LIN {X 0,Y 248.769,Z 1005.47,A -85,B 0,C 180,E1 11445.151,E2 11445.151} C_VEL
LIN {X 0,Y 248.089,Z 1009.313,A -85,B 0,C 180,E1 11439.986,E2 11439.986} C_VEL
LIN {X 0,Y 247.98,Z 1011.318,A -85,B 0,C 180,E1 11435.56,E2 11435.56} C_VEL
LIN {X 0,Y 248.003,Z 1012.187,A -85,B 0,C 180,E1 11431.393,E2 11431.393} C_VEL
LIN {X 0,Y 247.976,Z 1011.971,A -85,B 0,C 180,E1 11426.771,E2 11426.771} C_VEL
LIN {X 0,Y 247.994,Z 1010.436,A -85,B 0,C 180,E1 11422.362,E2 11422.362} C_VEL
LIN {X 0,Y 248.248,Z 1007.938,A -85,B 0,C 180,E1 11418.154,E2 11418.154} C_VEL
LIN {X 0,Y 249.171,Z 1003.742,A -85,B 0,C 180,E1 11413.215,E2 11413.215} C_VEL
LIN {X 0,Y 251.144,Z 997.579,A -85,B 0,C 180,E1 11408.065,E2 11408.065} C_VEL
LIN {X 0,Y 254.45,Z 989.685,A -85,B 0,C 180,E1 11402.891,E2 11402.891} C_VEL
LIN {X 0,Y 258.825,Z 980.598,A -85,B 0,C 180,E1 11398.196,E2 11398.196} C_VEL
LIN {X 0,Y 264.874,Z 969.114,A -85,B 0,C 180,E1 11393.396,E2 11393.396} C_VEL
LIN {X 0,Y 271.46,Z 957.155,A -85,B 0,C 180,E1 11389.323,E2 11389.323} C_VEL
LIN {X 0,Y 279.185,Z 943.15,A -85,B 0,C 180,E1 11385.428,E2 11385.428} C_VEL
LIN {X 0,Y 287.538,Z 927.889,A -85,B 0,C 180,E1 11381.926,E2 11381.926} C_VEL
LIN {X 0,Y 296.257,Z 911.009,A -85,B 0,C 180,E1 11378.787,E2 11378.787} C_VEL
LIN {X 0,Y 305.508,Z 892.125,A -85,B 0,C 180,E1 11375.916,E2 11375.916} C_VEL
LIN {X 0,Y 313.91,Z 873.62,A -85,B 0,C 180,E1 11373.613,E2 11373.613} C_VEL
LIN {X 0,Y 321.806,Z 854.322,A -85,B 0,C 180,E1 11371.658,E2 11371.658} C_VEL
LIN {X 0,Y 329.269,Z 834.233,A -85,B 0,C 180,E1 11369.98,E2 11369.98} C_VEL
LIN {X 0,Y 335.891,Z 813.522,A -85,B 0,C 180,E1 11368.596,E2 11368.596} C_VEL
LIN {X 0,Y 341.852,Z 792.201,A -85,B 0,C 180,E1 11367.446,E2 11367.446} C_VEL
LIN {X 0,Y 346.788,Z 770.459,A -85,B 0,C 180,E1 11366.544,E2 11366.544} C_VEL
LIN {X 0,Y 351.119,Z 746.303,A -85,B 0,C 180,E1 11365.792,E2 11365.792} C_VEL
LIN {X 0,Y 353.796,Z 723.704,A -85,B 0,C 180,E1 11365.251,E2 11365.251} C_VEL
LIN {X 0,Y 369.048,Z 537.52,A -85,B 0,C 180,E1 11361.492,E2 11361.492} C_VEL
LIN {X 0,Y 363.248,Z 527.675,A -85,B 0,C 180,E1 11359.036,E2 11359.036} C_VEL
LIN {X 0,Y 357.672,Z 518.823,A -85,B 0,C 180,E1 11356.441,E2 11356.441} C_VEL
LIN {X 0,Y 350.936,Z 509.322,A -85,B 0,C 180,E1 11352.923,E2 11352.923} C_VEL
LIN {X 0,Y 346.797,Z 503.841,A -85,B 0,C 180,E1 11350.464,E2 11350.464} C_VEL
LIN {X 0,Y 343.075,Z 498.85,A -85,B 0,C 180,E1 11347.957,E2 11347.957} C_VEL
LIN {X 0,Y 339.371,Z 493.892,A -85,B 0,C 180,E1 11345.07,E2 11345.07} C_VEL
LIN {X 0,Y 336.137,Z 489.935,A -85,B 0,C 180,E1 11342.114,E2 11342.114} C_VEL
LIN {X 0,Y 335.121,Z 488.35,A -85,B 0,C 180,E1 11341.025,E2 11341.025} C_VEL
LIN {X 0,Y 331.973,Z 484.932,A -85,B 0,C 180,E1 11337.151,E2 11337.151} C_VEL
LIN {X 0,Y 330.953,Z 482.618,A -85,B 0,C 180,E1 11335.32,E2 11335.32} C_VEL
LIN {X 0,Y 328.272,Z 480.723,A -85,B 0,C 180,E1 11328.224,E2 11328.224} C_VEL
LIN {X 0,Y 328.227,Z 480.713,A -85,B 0,C 180,E1 11323.36,E2 11323.36} C_VEL
LIN {X 0,Y 330.956,Z 482.61,A -85,B 0,C 180,E1 11315.929,E2 11315.929} C_VEL
LIN {X 0,Y 333.571,Z 487.051,A -85,B 0,C 180,E1 11311.926,E2 11311.926} C_VEL
LIN {X 0,Y 335.647,Z 488.946,A -85,B 0,C 180,E1 11309.683,E2 11309.683} C_VEL
LIN {X 0,Y 338.748,Z 493.298,A -85,B 0,C 180,E1 11306.701,E2 11306.701} C_VEL
LIN {X 0,Y 340.159,Z 494.956,A -85,B 0,C 180,E1 11305.539,E2 11305.539} C_VEL
LIN {X 0,Y 344.371,Z 500.521,A -85,B 0,C 180,E1 11302.421,E2 11302.421} C_VEL
LIN {X 0,Y 348.619,Z 506.23,A -85,B 0,C 180,E1 11299.71,E2 11299.71} C_VEL
LIN {X 0,Y 352.841,Z 512.104,A -85,B 0,C 180,E1 11297.314,E2 11297.314} C_VEL
LIN {X 0,Y 358.459,Z 519.986,A -85,B 0,C 180,E1 11294.489,E2 11294.489} C_VEL
LIN {X 0,Y 365.158,Z 529.934,A -85,B 0,C 180,E1 11291.493,E2 11291.493} C_VEL
LIN {X 0,Y 368.682,Z 535.581,A -85,B 0,C 180,E1 11290.037,E2 11290.037} C_VEL
LIN {X 0,Y 353.501,Z 718.347,A -85,B 0,C 180,E1 11286.344,E2 11286.344} C_VEL
LIN {X 0,Y 350.103,Z 742.254,A -85,B 0,C 180,E1 11285.689,E2 11285.689} C_VEL
LIN {X 0,Y 345.867,Z 764.626,A -85,B 0,C 180,E1 11284.859,E2 11284.859} C_VEL
LIN {X 0,Y 340.555,Z 786.357,A -85,B 0,C 180,E1 11283.797,E2 11283.797} C_VEL
LIN {X 0,Y 334.282,Z 808.106,A -85,B 0,C 180,E1 11282.465,E2 11282.465} C_VEL
LIN {X 0,Y 327.833,Z 827.172,A -85,B 0,C 180,E1 11281.019,E2 11281.019} C_VEL
LIN {X 0,Y 319.891,Z 847.961,A -85,B 0,C 180,E1 11279.098,E2 11279.098} C_VEL
LIN {X 0,Y 312.126,Z 866.095,A -85,B 0,C 180,E1 11277.05,E2 11277.05} C_VEL
LIN {X 0,Y 303.456,Z 884.529,A -85,B 0,C 180,E1 11274.522,E2 11274.522} C_VEL
LIN {X 0,Y 295.342,Z 900.625,A -85,B 0,C 180,E1 11271.856,E2 11271.856} C_VEL
LIN {X 0,Y 286.891,Z 916.302,A -85,B 0,C 180,E1 11268.694,E2 11268.694} C_VEL
LIN {X 0,Y 278.817,Z 930.785,A -85,B 0,C 180,E1 11265.169,E2 11265.169} C_VEL
LIN {X 0,Y 271.276,Z 943.789,A -85,B 0,C 180,E1 11261.258,E2 11261.258} C_VEL
LIN {X 0,Y 264.24,Z 956.093,A -85,B 0,C 180,E1 11256.729,E2 11256.729} C_VEL
LIN {X 0,Y 259.012,Z 965.539,A -85,B 0,C 180,E1 11252.427,E2 11252.427} C_VEL
LIN {X 0,Y 254.363,Z 974.561,A -85,B 0,C 180,E1 11247.29,E2 11247.29} C_VEL
LIN {X 0,Y 251.266,Z 981.545,A -85,B 0,C 180,E1 11242.247,E2 11242.247} C_VEL
LIN {X 0,Y 249.362,Z 986.687,A -85,B 0,C 180,E1 11237.253,E2 11237.253} C_VEL
LIN {X 0,Y 248.437,Z 990.344,A -85,B 0,C 180,E1 11232.425,E2 11232.425} C_VEL
LIN {X 0,Y 248.066,Z 992.682,A -85,B 0,C 180,E1 11227.373,E2 11227.373} C_VEL
LIN {X 0,Y 247.999,Z 993.543,A -85,B 0,C 180,E1 11223.409,E2 11223.409} C_VEL
LIN {X 0,Y 248.016,Z 993.556,A -85,B 0,C 180,E1 11219.465,E2 11219.465} C_VEL
LIN {X 0,Y 248.186,Z 992.42,A -85,B 0,C 180,E1 11214.534,E2 11214.534} C_VEL
LIN {X 0,Y 248.752,Z 989.887,A -85,B 0,C 180,E1 11209.667,E2 11209.667} C_VEL
LIN {X 0,Y 250.122,Z 986.016,A -85,B 0,C 180,E1 11204.631,E2 11204.631} C_VEL
LIN {X 0,Y 252.616,Z 980.364,A -85,B 0,C 180,E1 11199.475,E2 11199.475} C_VEL
LIN {X 0,Y 256.451,Z 973.276,A -85,B 0,C 180,E1 11194.426,E2 11194.426} C_VEL
LIN {X 0,Y 259.234,Z 968.524,A -85,B 0,C 180,E1 11191.656,E2 11191.656} C_VEL
LIN {X 0,Y 260.09,Z 965.887,A -85,B 0,C 180,E1 11190.056,E2 11190.056} C_VEL
LIN {X 0,Y 259.629,Z 958.618,A -85,B 0,C 180,E1 11185.651,E2 11185.651} C_VEL
LIN {X 0,Y 260.902,Z 955.846,A -85,B 0,C 180,E1 11184.347,E2 11184.347} C_VEL
LIN {X 0,Y 268.781,Z 944.21,A -85,B 0,C 180,E1 11180.014,E2 11180.014} C_VEL
LIN {X 0,Y 278.131,Z 930.421,A -85,B 0,C 180,E1 11175.856,E2 11175.856} C_VEL
LIN {X 0,Y 286.879,Z 917.067,A -85,B 0,C 180,E1 11172.591,E2 11172.591} C_VEL
LIN {X 0,Y 297.228,Z 900.535,A -85,B 0,C 180,E1 11169.293,E2 11169.293} C_VEL
LIN {X 0,Y 307.195,Z 883.613,A -85,B 0,C 180,E1 11166.542,E2 11166.542} C_VEL
LIN {X 0,Y 316.877,Z 865.511,A -85,B 0,C 180,E1 11164.163,E2 11164.163} C_VEL
LIN {X 0,Y 326.234,Z 846.492,A -85,B 0,C 180,E1 11162.108,E2 11162.108} C_VEL
LIN {X 0,Y 334.593,Z 827.332,A -85,B 0,C 180,E1 11160.429,E2 11160.429} C_VEL
LIN {X 0,Y 342.772,Z 806.039,A -85,B 0,C 180,E1 11158.914,E2 11158.914} C_VEL
LIN {X 0,Y 349.225,Z 786.548,A -85,B 0,C 180,E1 11157.799,E2 11157.799} C_VEL
LIN {X 0,Y 355.509,Z 763.656,A -85,B 0,C 180,E1 11156.762,E2 11156.762} C_VEL
LIN {X 0,Y 359.938,Z 743.618,A -85,B 0,C 180,E1 11156.062,E2 11156.062} C_VEL
LIN {X 0,Y 363.887,Z 719.388,A -85,B 0,C 180,E1 11155.435,E2 11155.435} C_VEL
LIN {X 0,Y 383.022,Z 548.711,A -85,B 0,C 180,E1 11151.972,E2 11151.972} C_VEL
LIN {X 0,Y 381.952,Z 546.067,A -85,B 0,C 180,E1 11150.508,E2 11150.508} C_VEL
LIN {X 0,Y 381.336,Z 544.156,A -85,B 0,C 180,E1 11149.272,E2 11149.272} C_VEL
LIN {X 0,Y 380.669,Z 542.357,A -85,B 0,C 180,E1 11146.172,E2 11146.172} C_VEL
LIN {X 0,Y 381.477,Z 544.535,A -85,B 0,C 180,E1 11142.851,E2 11142.851} C_VEL
LIN {X 0,Y 382.931,Z 548.576,A -85,B 0,C 180,E1 11140.555,E2 11140.555} C_VEL
LIN {X 0,Y 383.035,Z 549.077,A -85,B 0,C 180,E1 11140.399,E2 11140.399} C_VEL
LIN {X 0,Y 362.692,Z 730.721,A -85,B 0,C 180,E1 11136.705,E2 11136.705} C_VEL
LIN {X 0,Y 358.409,Z 754.445,A -85,B 0,C 180,E1 11136.093,E2 11136.093} C_VEL
LIN {X 0,Y 352.927,Z 777.381,A -85,B 0,C 180,E1 11135.333,E2 11135.333} C_VEL
LIN {X 0,Y 346.699,Z 798.517,A -85,B 0,C 180,E1 11134.399,E2 11134.399} C_VEL
LIN {X 0,Y 339.018,Z 820.594,A -85,B 0,C 180,E1 11133.152,E2 11133.152} C_VEL
LIN {X 0,Y 331.343,Z 839.865,A -85,B 0,C 180,E1 11131.787,E2 11131.787} C_VEL
LIN {X 0,Y 321.816,Z 861.077,A -85,B 0,C 180,E1 11129.921,E2 11129.921} C_VEL
LIN {X 0,Y 312.718,Z 879.494,A -85,B 0,C 180,E1 11127.925,E2 11127.925} C_VEL
LIN {X 0,Y 302.497,Z 898.396,A -85,B 0,C 180,E1 11125.396,E2 11125.396} C_VEL
LIN {X 0,Y 292.361,Z 916.045,A -85,B 0,C 180,E1 11122.502,E2 11122.502} C_VEL
LIN {X 0,Y 282.55,Z 932.109,A -85,B 0,C 180,E1 11119.232,E2 11119.232} C_VEL
LIN {X 0,Y 272.441,Z 948.205,A -85,B 0,C 180,E1 11115.201,E2 11115.201} C_VEL
LIN {X 0,Y 263.857,Z 961.864,A -85,B 0,C 180,E1 11110.969,E2 11110.969} C_VEL
LIN {X 0,Y 256.394,Z 973.776,A -85,B 0,C 180,E1 11106.359,E2 11106.359} C_VEL
LIN {X 0,Y 250.204,Z 984.397,A -85,B 0,C 180,E1 11101.306,E2 11101.306} C_VEL
LIN {X 0,Y 245.794,Z 992.731,A -85,B 0,C 180,E1 11096.328,E2 11096.328} C_VEL
LIN {X 0,Y 242.454,Z 1000.349,A -85,B 0,C 180,E1 11090.527,E2 11090.527} C_VEL
LIN {X 0,Y 240.859,Z 1005.238,A -85,B 0,C 180,E1 11085.621,E2 11085.621} C_VEL
LIN {X 0,Y 240.107,Z 1009.027,A -85,B 0,C 180,E1 11080.322,E2 11080.322} C_VEL
LIN {X 0,Y 239.985,Z 1011.028,A -85,B 0,C 180,E1 11075.746,E2 11075.746} C_VEL
LIN {X 0,Y 240.011,Z 1011.863,A -85,B 0,C 180,E1 11071.678,E2 11071.678} C_VEL
LIN {X 0,Y 239.993,Z 1011.753,A -85,B 0,C 180,E1 11067.381,E2 11067.381} C_VEL
LIN {X 0,Y 239.989,Z 1010.321,A -85,B 0,C 180,E1 11062.548,E2 11062.548} C_VEL
LIN {X 0,Y 240.269,Z 1007.717,A -85,B 0,C 180,E1 11057.936,E2 11057.936} C_VEL
LIN {X 0,Y 241.247,Z 1003.603,A -85,B 0,C 180,E1 11052.895,E2 11052.895} C_VEL
LIN {X 0,Y 243.357,Z 997.456,A -85,B 0,C 180,E1 11047.545,E2 11047.545} C_VEL
LIN {X 0,Y 246.843,Z 989.668,A -85,B 0,C 180,E1 11042.246,E2 11042.246} C_VEL
LIN {X 0,Y 251.412,Z 980.698,A -85,B 0,C 180,E1 11037.469,E2 11037.469} C_VEL
LIN {X 0,Y 257.831,Z 969.179,A -85,B 0,C 180,E1 11032.505,E2 11032.505} C_VEL
LIN {X 0,Y 264.721,Z 957.254,A -85,B 0,C 180,E1 11028.347,E2 11028.347} C_VEL
LIN {X 0,Y 272.787,Z 943.296,A -85,B 0,C 180,E1 11024.389,E2 11024.389} C_VEL
LIN {X 0,Y 281.465,Z 928.077,A -85,B 0,C 180,E1 11020.843,E2 11020.843} C_VEL
LIN {X 0,Y 290.227,Z 911.789,A -85,B 0,C 180,E1 11017.767,E2 11017.767} C_VEL
LIN {X 0,Y 299.168,Z 894.342,A -85,B 0,C 180,E1 11015.046,E2 11015.046} C_VEL
LIN {X 0,Y 307.445,Z 876.72,A -85,B 0,C 180,E1 11012.802,E2 11012.802} C_VEL
LIN {X 0,Y 316.512,Z 855.618,A -85,B 0,C 180,E1 11010.605,E2 11010.605} C_VEL
LIN {X 0,Y 323.951,Z 836.249,A -85,B 0,C 180,E1 11008.969,E2 11008.969} C_VEL
LIN {X 0,Y 331.096,Z 814.921,A -85,B 0,C 180,E1 11007.518,E2 11007.518} C_VEL
LIN {X 0,Y 337.055,Z 794.388,A -85,B 0,C 180,E1 11006.396,E2 11006.396} C_VEL
LIN {X 0,Y 342.358,Z 772.067,A -85,B 0,C 180,E1 11005.453,E2 11005.453} C_VEL
LIN {X 0,Y 346.782,Z 748.869,A -85,B 0,C 180,E1 11004.715,E2 11004.715} C_VEL
LIN {X 0,Y 349.714,Z 725.457,A -85,B 0,C 180,E1 11004.149,E2 11004.149} C_VEL
LIN {X 0,Y 365.239,Z 542.064,A -85,B 0,C 180,E1 11000.451,E2 11000.451} C_VEL
LIN {X 0,Y 358.467,Z 530.554,A -85,B 0,C 180,E1 10997.406,E2 10997.406} C_VEL
LIN {X 0,Y 352.701,Z 521.833,A -85,B 0,C 180,E1 10994.529,E2 10994.529} C_VEL
LIN {X 0,Y 345.834,Z 512.201,A -85,B 0,C 180,E1 10990.578,E2 10990.578} C_VEL
LIN {X 0,Y 341.407,Z 506.37,A -85,B 0,C 180,E1 10987.572,E2 10987.572} C_VEL
LIN {X 0,Y 337.873,Z 501.562,A -85,B 0,C 180,E1 10984.752,E2 10984.752} C_VEL
LIN {X 0,Y 334.644,Z 497.443,A -85,B 0,C 180,E1 10981.711,E2 10981.711} C_VEL
LIN {X 0,Y 333.852,Z 496.194,A -85,B 0,C 180,E1 10980.857,E2 10980.857} C_VEL
LIN {X 0,Y 330.703,Z 492.674,A -85,B 0,C 180,E1 10976.88,E2 10976.88} C_VEL
LIN {X 0,Y 329.743,Z 490.493,A -85,B 0,C 180,E1 10975.129,E2 10975.129} C_VEL
LIN {X 0,Y 327.145,Z 488.625,A -85,B 0,C 180,E1 10968.004,E2 10968.004} C_VEL
LIN {X 0,Y 327.171,Z 488.653,A -85,B 0,C 180,E1 10963.122,E2 10963.122} C_VEL
LIN {X 0,Y 329.859,Z 490.536,A -85,B 0,C 180,E1 10955.939,E2 10955.939} C_VEL
LIN {X 0,Y 331.974,Z 494.463,A -85,B 0,C 180,E1 10952.56,E2 10952.56} C_VEL
LIN {X 0,Y 334.299,Z 496.722,A -85,B 0,C 180,E1 10949.935,E2 10949.935} C_VEL
LIN {X 0,Y 337.446,Z 501.142,A -85,B 0,C 180,E1 10946.86,E2 10946.86} C_VEL
LIN {X 0,Y 338.732,Z 502.759,A -85,B 0,C 180,E1 10945.773,E2 10945.773} C_VEL
LIN {X 0,Y 342.741,Z 508.121,A -85,B 0,C 180,E1 10942.747,E2 10942.747} C_VEL
LIN {X 0,Y 347.017,Z 513.985,A -85,B 0,C 180,E1 10939.965,E2 10939.965} C_VEL
LIN {X 0,Y 351.105,Z 519.747,A -85,B 0,C 180,E1 10937.607,E2 10937.607} C_VEL
LIN {X 0,Y 356.737,Z 527.858,A -85,B 0,C 180,E1 10934.723,E2 10934.723} C_VEL
LIN {X 0,Y 363.169,Z 537.543,A -85,B 0,C 180,E1 10931.804,E2 10931.804} C_VEL
LIN {X 0,Y 364.841,Z 540.526,A -85,B 0,C 180,E1 10931.073,E2 10931.073} C_VEL
LIN {X 0,Y 349.587,Z 718.787,A -85,B 0,C 180,E1 10927.479,E2 10927.479} C_VEL
LIN {X 0,Y 346.106,Z 742.652,A -85,B 0,C 180,E1 10926.828,E2 10926.828} C_VEL
LIN {X 0,Y 341.787,Z 764.94,A -85,B 0,C 180,E1 10926.007,E2 10926.007} C_VEL
LIN {X 0,Y 336.502,Z 786.077,A -85,B 0,C 180,E1 10924.984,E2 10924.984} C_VEL
LIN {X 0,Y 330.381,Z 806.998,A -85,B 0,C 180,E1 10923.726,E2 10923.726} C_VEL
LIN {X 0,Y 323.418,Z 827.076,A -85,B 0,C 180,E1 10922.22,E2 10922.22} C_VEL
LIN {X 0,Y 315.469,Z 847.42,A -85,B 0,C 180,E1 10920.358,E2 10920.358} C_VEL
LIN {X 0,Y 307.516,Z 865.523,A -85,B 0,C 180,E1 10918.332,E2 10918.332} C_VEL
LIN {X 0,Y 298.262,Z 884.679,A -85,B 0,C 180,E1 10915.722,E2 10915.722} C_VEL
LIN {X 0,Y 289.589,Z 901.284,A -85,B 0,C 180,E1 10912.957,E2 10912.957} C_VEL
LIN {X 0,Y 280.813,Z 916.911,A -85,B 0,C 180,E1 10909.763,E2 10909.763} C_VEL
LIN {X 0,Y 272.418,Z 931.375,A -85,B 0,C 180,E1 10906.19,E2 10906.19} C_VEL
LIN {X 0,Y 264.905,Z 943.764,A -85,B 0,C 180,E1 10902.417,E2 10902.417} C_VEL
LIN {X 0,Y 257.789,Z 955.628,A -85,B 0,C 180,E1 10898.019,E2 10898.019} C_VEL
LIN {X 0,Y 252.156,Z 965.167,A -85,B 0,C 180,E1 10893.63,E2 10893.63} C_VEL
LIN {X 0,Y 247.076,Z 974.436,A -85,B 0,C 180,E1 10888.314,E2 10888.314} C_VEL
LIN {X 0,Y 243.825,Z 981.138,A -85,B 0,C 180,E1 10883.4,E2 10883.4} C_VEL
LIN {X 0,Y 241.605,Z 986.675,A -85,B 0,C 180,E1 10878.051,E2 10878.051} C_VEL
LIN {X 0,Y 240.562,Z 990.23,A -85,B 0,C 180,E1 10873.327,E2 10873.327} C_VEL
LIN {X 0,Y 240.103,Z 992.77,A -85,B 0,C 180,E1 10868.226,E2 10868.226} C_VEL
LIN {X 0,Y 240.002,Z 993.802,A -85,B 0,C 180,E1 10863.787,E2 10863.787} C_VEL
LIN {X 0,Y 240.014,Z 993.89,A -85,B 0,C 180,E1 10859.724,E2 10859.724} C_VEL
LIN {X 0,Y 240.142,Z 993.034,A -85,B 0,C 180,E1 10855.214,E2 10855.214} C_VEL
LIN {X 0,Y 240.736,Z 990.603,A -85,B 0,C 180,E1 10849.839,E2 10849.839} C_VEL
LIN {X 0,Y 242.012,Z 987.115,A -85,B 0,C 180,E1 10844.95,E2 10844.95} C_VEL
LIN {X 0,Y 244.702,Z 981.448,A -85,B 0,C 180,E1 10839.298,E2 10839.298} C_VEL
LIN {X 0,Y 248.488,Z 974.816,A -85,B 0,C 180,E1 10834.287,E2 10834.287} C_VEL
LIN {X 0,Y 254.06,Z 965.972,A -85,B 0,C 180,E1 10829.1,E2 10829.1} C_VEL
LIN {X 0,Y 260.902,Z 955.846,A -85,B 0,C 180,E1 10824.347,E2 10824.347} C_VEL
LIN {X 0,Y 262.433,Z 952.59,A -85,B 0,C 180,E1 10822.838,E2 10822.838} C_VEL
LIN {X 0,Y 263.812,Z 944.549,A -85,B 0,C 180,E1 10818.828,E2 10818.828} C_VEL
LIN {X 0,Y 265.766,Z 940.73,A -85,B 0,C 180,E1 10817.428,E2 10817.428} C_VEL
LIN {X 0,Y 275.039,Z 927.564,A -85,B 0,C 180,E1 10813.669,E2 10813.669} C_VEL
LIN {X 0,Y 285.568,Z 912.095,A -85,B 0,C 180,E1 10810.083,E2 10810.083} C_VEL
LIN {X 0,Y 295.441,Z 896.734,A -85,B 0,C 180,E1 10807.194,E2 10807.194} C_VEL
LIN {X 0,Y 305.947,Z 879.096,A -85,B 0,C 180,E1 10804.499,E2 10804.499} C_VEL
LIN {X 0,Y 316.202,Z 860.436,A -85,B 0,C 180,E1 10802.182,E2 10802.182} C_VEL
LIN {X 0,Y 325.562,Z 841.261,A -85,B 0,C 180,E1 10800.265,E2 10800.265} C_VEL
LIN {X 0,Y 335.085,Z 819.376,A -85,B 0,C 180,E1 10798.497,E2 10798.497} C_VEL
LIN {X 0,Y 342.621,Z 799.315,A -85,B 0,C 180,E1 10797.201,E2 10797.201} C_VEL
LIN {X 0,Y 349.646,Z 777.241,A -85,B 0,C 180,E1 10796.065,E2 10796.065} C_VEL
LIN {X 0,Y 355.517,Z 754.778,A -85,B 0,C 180,E1 10795.168,E2 10795.168} C_VEL
LIN {X 0,Y 360.058,Z 731.664,A -85,B 0,C 180,E1 10794.488,E2 10794.488} C_VEL
LIN {X 0,Y 363.834,Z 703.722,A -85,B 0,C 180,E1 10793.875,E2 10793.875} C_VEL
LIN {X 0,Y 381.097,Z 554.779,A -85,B 0,C 180,E1 10790.905,E2 10790.905} C_VEL
LIN {X 0,Y 380.067,Z 551.885,A -85,B 0,C 180,E1 10788.929,E2 10788.929} C_VEL
LIN {X 0,Y 379.576,Z 550.299,A -85,B 0,C 180,E1 10786.131,E2 10786.131} C_VEL
LIN {X 0,Y 380.272,Z 552.394,A -85,B 0,C 180,E1 10783.032,E2 10783.032} C_VEL
LIN {X 0,Y 381.098,Z 555.155,A -85,B 0,C 180,E1 10781.472,E2 10781.472} C_VEL
LIN {X 0,Y 360.729,Z 730.116,A -85,B 0,C 180,E1 10777.95,E2 10777.95} C_VEL
LIN {X 0,Y 356.328,Z 753.84,A -85,B 0,C 180,E1 10777.35,E2 10777.35} C_VEL
LIN {X 0,Y 350.574,Z 777.27,A -85,B 0,C 180,E1 10776.592,E2 10776.592} C_VEL
LIN {X 0,Y 344.436,Z 797.488,A -85,B 0,C 180,E1 10775.722,E2 10775.722} C_VEL
LIN {X 0,Y 336.695,Z 819.223,A -85,B 0,C 180,E1 10774.531,E2 10774.531} C_VEL
LIN {X 0,Y 329.156,Z 837.633,A -85,B 0,C 180,E1 10773.269,E2 10773.269} C_VEL
LIN {X 0,Y 319.676,Z 858.365,A -85,B 0,C 180,E1 10771.516,E2 10771.516} C_VEL
LIN {X 0,Y 310.487,Z 876.364,A -85,B 0,C 180,E1 10769.631,E2 10769.631} C_VEL
LIN {X 0,Y 299.562,Z 896.079,A -85,B 0,C 180,E1 10767.088,E2 10767.088} C_VEL
LIN {X 0,Y 289.251,Z 913.346,A -85,B 0,C 180,E1 10764.331,E2 10764.331} C_VEL
LIN {X 0,Y 278.846,Z 929.712,A -85,B 0,C 180,E1 10761.094,E2 10761.094} C_VEL
LIN {X 0,Y 268.928,Z 944.9,A -85,B 0,C 180,E1 10757.412,E2 10757.412} C_VEL
LIN {X 0,Y 259.819,Z 958.378,A -85,B 0,C 180,E1 10753.339,E2 10753.339} C_VEL
LIN {X 0,Y 251.088,Z 971.538,A -85,B 0,C 180,E1 10748.411,E2 10748.411} C_VEL
LIN {X 0,Y 244.45,Z 981.996,A -85,B 0,C 180,E1 10743.524,E2 10743.524} C_VEL
LIN {X 0,Y 239.141,Z 991.047,A -85,B 0,C 180,E1 10738.201,E2 10738.201} C_VEL
LIN {X 0,Y 235.474,Z 998.457,A -85,B 0,C 180,E1 10732.738,E2 10732.738} C_VEL
LIN {X 0,Y 233.26,Z 1004.066,A -85,B 0,C 180,E1 10727.211,E2 10727.211} C_VEL
LIN {X 0,Y 232.278,Z 1007.877,A -85,B 0,C 180,E1 10722.184,E2 10722.184} C_VEL
LIN {X 0,Y 231.985,Z 1010.435,A -85,B 0,C 180,E1 10716.939,E2 10716.939} C_VEL
LIN {X 0,Y 232.002,Z 1011.484,A -85,B 0,C 180,E1 10712.477,E2 10712.477} C_VEL
LIN {X 0,Y 232.016,Z 1011.532,A -85,B 0,C 180,E1 10708.279,E2 10708.279} C_VEL
LIN {X 0,Y 232,Z 1010.512,A -85,B 0,C 180,E1 10703.574,E2 10703.574} C_VEL
LIN {X 0,Y 232.229,Z 1007.911,A -85,B 0,C 180,E1 10698.333,E2 10698.333} C_VEL
LIN {X 0,Y 233.042,Z 1004.316,A -85,B 0,C 180,E1 10693.559,E2 10693.559} C_VEL
LIN {X 0,Y 235.074,Z 998.6,A -85,B 0,C 180,E1 10688.005,E2 10688.005} C_VEL
LIN {X 0,Y 238.295,Z 991.505,A -85,B 0,C 180,E1 10682.793,E2 10682.793} C_VEL
LIN {X 0,Y 243.493,Z 981.768,A -85,B 0,C 180,E1 10677.188,E2 10677.188} C_VEL
LIN {X 0,Y 249.485,Z 971.538,A -85,B 0,C 180,E1 10672.481,E2 10672.481} C_VEL
LIN {X 0,Y 256.847,Z 959.294,A -85,B 0,C 180,E1 10667.978,E2 10667.978} C_VEL
LIN {X 0,Y 265.078,Z 945.823,A -85,B 0,C 180,E1 10663.921,E2 10663.921} C_VEL
LIN {X 0,Y 273.407,Z 931.745,A -85,B 0,C 180,E1 10660.49,E2 10660.49} C_VEL
LIN {X 0,Y 282.74,Z 915.393,A -85,B 0,C 180,E1 10657.207,E2 10657.207} C_VEL
LIN {X 0,Y 291.902,Z 898.264,A -85,B 0,C 180,E1 10654.414,E2 10654.414} C_VEL
LIN {X 0,Y 301.369,Z 879.119,A -85,B 0,C 180,E1 10651.875,E2 10651.875} C_VEL
LIN {X 0,Y 310.288,Z 859.446,A -85,B 0,C 180,E1 10649.751,E2 10649.751} C_VEL
LIN {X 0,Y 318.231,Z 839.499,A -85,B 0,C 180,E1 10648.024,E2 10648.024} C_VEL
LIN {X 0,Y 325.764,Z 818.254,A -85,B 0,C 180,E1 10646.529,E2 10646.529} C_VEL
LIN {X 0,Y 331.958,Z 797.71,A -85,B 0,C 180,E1 10645.382,E2 10645.382} C_VEL
LIN {X 0,Y 338.064,Z 773.433,A -85,B 0,C 180,E1 10644.33,E2 10644.33} C_VEL
LIN {X 0,Y 342.572,Z 750.795,A -85,B 0,C 180,E1 10643.603,E2 10643.603} C_VEL
LIN {X 0,Y 345.746,Z 727.144,A -85,B 0,C 180,E1 10643.022,E2 10643.022} C_VEL
LIN {X 0,Y 361.488,Z 546.632,A -85,B 0,C 180,E1 10639.384,E2 10639.384} C_VEL
LIN {X 0,Y 354.884,Z 535.513,A -85,B 0,C 180,E1 10636.279,E2 10636.279} C_VEL
LIN {X 0,Y 349.392,Z 527.419,A -85,B 0,C 180,E1 10633.402,E2 10633.402} C_VEL
LIN {X 0,Y 344.1,Z 519.702,A -85,B 0,C 180,E1 10630.209,E2 10630.209} C_VEL
LIN {X 0,Y 339.754,Z 513.887,A -85,B 0,C 180,E1 10627.184,E2 10627.184} C_VEL
LIN {X 0,Y 336.38,Z 509.23,A -85,B 0,C 180,E1 10624.432,E2 10624.432} C_VEL
LIN {X 0,Y 333.199,Z 505.063,A -85,B 0,C 180,E1 10621.375,E2 10621.375} C_VEL
LIN {X 0,Y 332.422,Z 503.922,A -85,B 0,C 180,E1 10620.516,E2 10620.516} C_VEL
LIN {X 0,Y 329.469,Z 500.478,A -85,B 0,C 180,E1 10616.66,E2 10616.66} C_VEL
LIN {X 0,Y 328.538,Z 498.367,A -85,B 0,C 180,E1 10614.936,E2 10614.936} C_VEL
LIN {X 0,Y 326.051,Z 496.547,A -85,B 0,C 180,E1 10607.963,E2 10607.963} C_VEL
LIN {X 0,Y 326.092,Z 496.583,A -85,B 0,C 180,E1 10603.064,E2 10603.064} C_VEL
LIN {X 0,Y 328.691,Z 498.533,A -85,B 0,C 180,E1 10596.039,E2 10596.039} C_VEL
LIN {X 0,Y 330.942,Z 502.552,A -85,B 0,C 180,E1 10592.467,E2 10592.467} C_VEL
LIN {X 0,Y 333.02,Z 504.637,A -85,B 0,C 180,E1 10590.105,E2 10590.105} C_VEL
LIN {X 0,Y 336.178,Z 509.017,A -85,B 0,C 180,E1 10586.992,E2 10586.992} C_VEL
LIN {X 0,Y 337.754,Z 511.28,A -85,B 0,C 180,E1 10585.631,E2 10585.631} C_VEL
LIN {X 0,Y 341.131,Z 515.736,A -85,B 0,C 180,E1 10583.068,E2 10583.068} C_VEL
LIN {X 0,Y 345.255,Z 521.486,A -85,B 0,C 180,E1 10580.325,E2 10580.325} C_VEL
LIN {X 0,Y 349.577,Z 527.671,A -85,B 0,C 180,E1 10577.789,E2 10577.789} C_VEL
LIN {X 0,Y 356.82,Z 538.263,A -85,B 0,C 180,E1 10574.105,E2 10574.105} C_VEL
LIN {X 0,Y 361.106,Z 545.305,A -85,B 0,C 180,E1 10572.132,E2 10572.132} C_VEL
LIN {X 0,Y 345.801,Z 718.994,A -85,B 0,C 180,E1 10568.641,E2 10568.641} C_VEL
LIN {X 0,Y 342.238,Z 742.868,A -85,B 0,C 180,E1 10567.995,E2 10567.995} C_VEL
LIN {X 0,Y 337.831,Z 765.075,A -85,B 0,C 180,E1 10567.185,E2 10567.185} C_VEL
LIN {X 0,Y 332.247,Z 786.874,A -85,B 0,C 180,E1 10566.137,E2 10566.137} C_VEL
LIN {X 0,Y 325.635,Z 808.689,A -85,B 0,C 180,E1 10564.82,E2 10564.82} C_VEL
LIN {X 0,Y 318.827,Z 827.812,A -85,B 0,C 180,E1 10563.385,E2 10563.385} C_VEL
LIN {X 0,Y 310.339,Z 848.807,A -85,B 0,C 180,E1 10561.454,E2 10561.454} C_VEL
LIN {X 0,Y 302.167,Z 866.82,A -85,B 0,C 180,E1 10559.423,E2 10559.423} C_VEL
LIN {X 0,Y 292.91,Z 885.29,A -85,B 0,C 180,E1 10556.883,E2 10556.883} C_VEL
LIN {X 0,Y 283.943,Z 901.914,A -85,B 0,C 180,E1 10554.101,E2 10554.101} C_VEL
LIN {X 0,Y 274.838,Z 917.522,A -85,B 0,C 180,E1 10550.879,E2 10550.879} C_VEL
LIN {X 0,Y 266.105,Z 931.936,A -85,B 0,C 180,E1 10547.26,E2 10547.26} C_VEL
LIN {X 0,Y 258.262,Z 944.315,A -85,B 0,C 180,E1 10543.424,E2 10543.424} C_VEL
LIN {X 0,Y 250.811,Z 956.156,A -85,B 0,C 180,E1 10538.937,E2 10538.937} C_VEL
LIN {X 0,Y 244.885,Z 965.681,A -85,B 0,C 180,E1 10534.442,E2 10534.442} C_VEL
LIN {X 0,Y 239.558,Z 974.817,A -85,B 0,C 180,E1 10529.036,E2 10529.036} C_VEL
LIN {X 0,Y 236.069,Z 981.587,A -85,B 0,C 180,E1 10523.915,E2 10523.915} C_VEL
LIN {X 0,Y 233.709,Z 987.081,A -85,B 0,C 180,E1 10518.393,E2 10518.393} C_VEL
LIN {X 0,Y 232.59,Z 990.644,A -85,B 0,C 180,E1 10513.466,E2 10513.466} C_VEL
LIN {X 0,Y 232.109,Z 993.102,A -85,B 0,C 180,E1 10508.249,E2 10508.249} C_VEL
LIN {X 0,Y 232.008,Z 994.118,A -85,B 0,C 180,E1 10503.641,E2 10503.641} C_VEL
LIN {X 0,Y 232.03,Z 994.184,A -85,B 0,C 180,E1 10499.43,E2 10499.43} C_VEL
LIN {X 0,Y 232.209,Z 993.231,A -85,B 0,C 180,E1 10494.451,E2 10494.451} C_VEL
LIN {X 0,Y 232.917,Z 990.675,A -85,B 0,C 180,E1 10488.936,E2 10488.936} C_VEL
LIN {X 0,Y 234.535,Z 986.858,A -85,B 0,C 180,E1 10483.545,E2 10483.545} C_VEL
LIN {X 0,Y 237.575,Z 981.151,A -85,B 0,C 180,E1 10477.914,E2 10477.914} C_VEL
LIN {X 0,Y 242.148,Z 973.961,A -85,B 0,C 180,E1 10472.466,E2 10472.466} C_VEL
LIN {X 0,Y 248.153,Z 965.122,A -85,B 0,C 180,E1 10467.345,E2 10467.345} C_VEL
LIN {X 0,Y 256.08,Z 954.067,A -85,B 0,C 180,E1 10462.256,E2 10462.256} C_VEL
LIN {X 0,Y 264.769,Z 942.105,A -85,B 0,C 180,E1 10457.878,E2 10457.878} C_VEL
LIN {X 0,Y 265.766,Z 940.73,A -85,B 0,C 180,E1 10457.428,E2 10457.428} C_VEL
LIN {X 0,Y 267.871,Z 936.83,A -85,B 0,C 180,E1 10456.058,E2 10456.058} C_VEL
LIN {X 0,Y 271.277,Z 926.965,A -85,B 0,C 180,E1 10452.126,E2 10452.126} C_VEL
LIN {X 0,Y 273.481,Z 923.223,A -85,B 0,C 180,E1 10451.067,E2 10451.067} C_VEL
LIN {X 0,Y 283.971,Z 908.203,A -85,B 0,C 180,E1 10447.805,E2 10447.805} C_VEL
LIN {X 0,Y 295.378,Z 890.789,A -85,B 0,C 180,E1 10444.758,E2 10444.758} C_VEL
LIN {X 0,Y 306.209,Z 872.934,A -85,B 0,C 180,E1 10442.239,E2 10442.239} C_VEL
LIN {X 0,Y 316.044,Z 854.818,A -85,B 0,C 180,E1 10440.182,E2 10440.182} C_VEL
LIN {X 0,Y 325.436,Z 835.903,A -85,B 0,C 180,E1 10438.416,E2 10438.416} C_VEL
LIN {X 0,Y 334.07,Z 815.891,A -85,B 0,C 180,E1 10436.912,E2 10436.912} C_VEL
LIN {X 0,Y 341.977,Z 794.939,A -85,B 0,C 180,E1 10435.641,E2 10435.641} C_VEL
LIN {X 0,Y 348.216,Z 775.257,A -85,B 0,C 180,E1 10434.686,E2 10434.686} C_VEL
LIN {X 0,Y 354.26,Z 752.041,A -85,B 0,C 180,E1 10433.808,E2 10433.808} C_VEL
LIN {X 0,Y 358.751,Z 729.252,A -85,B 0,C 180,E1 10433.175,E2 10433.175} C_VEL
LIN {X 0,Y 363.032,Z 696.631,A -85,B 0,C 180,E1 10432.49,E2 10432.49} C_VEL
LIN {X 0,Y 379.334,Z 561.226,A -85,B 0,C 180,E1 10429.829,E2 10429.829} C_VEL
LIN {X 0,Y 378.887,Z 559.716,A -85,B 0,C 180,E1 10428.739,E2 10428.739} C_VEL
LIN {X 0,Y 378.481,Z 558.245,A -85,B 0,C 180,E1 10426.09,E2 10426.09} C_VEL
LIN {X 0,Y 379.061,Z 560.198,A -85,B 0,C 180,E1 10423.243,E2 10423.243} C_VEL
LIN {X 0,Y 379.343,Z 561.503,A -85,B 0,C 180,E1 10422.552,E2 10422.552} C_VEL
LIN {X 0,Y 359.033,Z 729.569,A -85,B 0,C 180,E1 10419.211,E2 10419.211} C_VEL
LIN {X 0,Y 354.525,Z 753.212,A -85,B 0,C 180,E1 10418.627,E2 10418.627} C_VEL
LIN {X 0,Y 348.843,Z 775.986,A -85,B 0,C 180,E1 10417.915,E2 10417.915} C_VEL
LIN {X 0,Y 342.526,Z 796.251,A -85,B 0,C 180,E1 10417.075,E2 10417.075} C_VEL
LIN {X 0,Y 334.587,Z 818.07,A -85,B 0,C 180,E1 10415.922,E2 10415.922} C_VEL
LIN {X 0,Y 326.446,Z 837.303,A -85,B 0,C 180,E1 10414.636,E2 10414.636} C_VEL
LIN {X 0,Y 316.323,Z 858.65,A -85,B 0,C 180,E1 10412.854,E2 10412.854} C_VEL
LIN {X 0,Y 307.013,Z 876.207,A -85,B 0,C 180,E1 10411.034,E2 10411.034} C_VEL
LIN {X 0,Y 295.9,Z 895.497,A -85,B 0,C 180,E1 10408.57,E2 10408.57} C_VEL
LIN {X 0,Y 285.815,Z 911.717,A -85,B 0,C 180,E1 10406.013,E2 10406.013} C_VEL
LIN {X 0,Y 274.312,Z 929.075,A -85,B 0,C 180,E1 10402.625,E2 10402.625} C_VEL
LIN {X 0,Y 263.892,Z 944.258,A -85,B 0,C 180,E1 10398.944,E2 10398.944} C_VEL
LIN {X 0,Y 254.128,Z 957.928,A -85,B 0,C 180,E1 10394.778,E2 10394.778} C_VEL
LIN {X 0,Y 245.347,Z 970.385,A -85,B 0,C 180,E1 10390.09,E2 10390.09} C_VEL
LIN {X 0,Y 238.432,Z 980.44,A -85,B 0,C 180,E1 10385.366,E2 10385.366} C_VEL
LIN {X 0,Y 232.042,Z 990.486,A -85,B 0,C 180,E1 10379.428,E2 10379.428} C_VEL
LIN {X 0,Y 228.131,Z 997.601,A -85,B 0,C 180,E1 10374.062,E2 10374.062} C_VEL
LIN {X 0,Y 225.504,Z 1003.595,A -85,B 0,C 180,E1 10368.089,E2 10368.089} C_VEL
LIN {X 0,Y 224.364,Z 1007.44,A -85,B 0,C 180,E1 10362.882,E2 10362.882} C_VEL
LIN {X 0,Y 223.991,Z 1010.07,A -85,B 0,C 180,E1 10357.445,E2 10357.445} C_VEL
LIN {X 0,Y 223.997,Z 1011.158,A -85,B 0,C 180,E1 10352.822,E2 10352.822} C_VEL
LIN {X 0,Y 224.019,Z 1011.265,A -85,B 0,C 180,E1 10348.729,E2 10348.729} C_VEL
LIN {X 0,Y 223.995,Z 1010.468,A -85,B 0,C 180,E1 10344.372,E2 10344.372} C_VEL
LIN {X 0,Y 224.147,Z 1008.376,A -85,B 0,C 180,E1 10339.21,E2 10339.21} C_VEL
LIN {X 0,Y 224.985,Z 1004.564,A -85,B 0,C 180,E1 10333.721,E2 10333.721} C_VEL
LIN {X 0,Y 226.809,Z 999.596,A -85,B 0,C 180,E1 10328.458,E2 10328.458} C_VEL
LIN {X 0,Y 230.113,Z 992.542,A -85,B 0,C 180,E1 10322.865,E2 10322.865} C_VEL
LIN {X 0,Y 234.845,Z 984.103,A -85,B 0,C 180,E1 10317.568,E2 10317.568} C_VEL
LIN {X 0,Y 241.127,Z 973.678,A -85,B 0,C 180,E1 10312.454,E2 10312.454} C_VEL
LIN {X 0,Y 248.813,Z 961.612,A -85,B 0,C 180,E1 10307.68,E2 10307.68} C_VEL
LIN {X 0,Y 256.897,Z 948.871,A -85,B 0,C 180,E1 10303.633,E2 10303.633} C_VEL
LIN {X 0,Y 266.405,Z 933.611,A -85,B 0,C 180,E1 10299.713,E2 10299.713} C_VEL
LIN {X 0,Y 275.835,Z 917.878,A -85,B 0,C 180,E1 10296.431,E2 10296.431} C_VEL
LIN {X 0,Y 285.433,Z 900.658,A -85,B 0,C 180,E1 10293.534,E2 10293.534} C_VEL
LIN {X 0,Y 295.045,Z 882.152,A -85,B 0,C 180,E1 10290.992,E2 10290.992} C_VEL
LIN {X 0,Y 303.809,Z 863.48,A -85,B 0,C 180,E1 10288.92,E2 10288.92} C_VEL
LIN {X 0,Y 312.961,Z 841.761,A -85,B 0,C 180,E1 10286.972,E2 10286.972} C_VEL
LIN {X 0,Y 320.601,Z 821.161,A -85,B 0,C 180,E1 10285.491,E2 10285.491} C_VEL
LIN {X 0,Y 327.354,Z 799.728,A -85,B 0,C 180,E1 10284.273,E2 10284.273} C_VEL
LIN {X 0,Y 333.365,Z 777.188,A -85,B 0,C 180,E1 10283.265,E2 10283.265} C_VEL
LIN {X 0,Y 338.147,Z 754.262,A -85,B 0,C 180,E1 10282.513,E2 10282.513} C_VEL
LIN {X 0,Y 341.882,Z 728.861,A -85,B 0,C 180,E1 10281.873,E2 10281.873} C_VEL
LIN {X 0,Y 357.862,Z 551.428,A -85,B 0,C 180,E1 10278.319,E2 10278.319} C_VEL
LIN {X 0,Y 351.945,Z 541.378,A -85,B 0,C 180,E1 10275.404,E2 10275.404} C_VEL
LIN {X 0,Y 345.562,Z 531.794,A -85,B 0,C 180,E1 10271.854,E2 10271.854} C_VEL
LIN {X 0,Y 341.367,Z 526.011,A -85,B 0,C 180,E1 10269.185,E2 10269.185} C_VEL
LIN {X 0,Y 338.196,Z 521.522,A -85,B 0,C 180,E1 10266.876,E2 10266.876} C_VEL
LIN {X 0,Y 334.871,Z 516.891,A -85,B 0,C 180,E1 10264.109,E2 10264.109} C_VEL
LIN {X 0,Y 331.691,Z 512.537,A -85,B 0,C 180,E1 10260.949,E2 10260.949} C_VEL
LIN {X 0,Y 330.701,Z 511.396,A -85,B 0,C 180,E1 10259.826,E2 10259.826} C_VEL
LIN {X 0,Y 327.955,Z 507.728,A -85,B 0,C 180,E1 10255.978,E2 10255.978} C_VEL
LIN {X 0,Y 327.311,Z 506.226,A -85,B 0,C 180,E1 10254.697,E2 10254.697} C_VEL
LIN {X 0,Y 324.929,Z 504.451,A -85,B 0,C 180,E1 10247.741,E2 10247.741} C_VEL
LIN {X 0,Y 325.012,Z 504.519,A -85,B 0,C 180,E1 10243.006,E2 10243.006} C_VEL
LIN {X 0,Y 327.483,Z 506.397,A -85,B 0,C 180,E1 10236.232,E2 10236.232} C_VEL
LIN {X 0,Y 329.773,Z 510.469,A -85,B 0,C 180,E1 10232.557,E2 10232.557} C_VEL
LIN {X 0,Y 331.657,Z 512.388,A -85,B 0,C 180,E1 10230.368,E2 10230.368} C_VEL
LIN {X 0,Y 334.952,Z 516.93,A -85,B 0,C 180,E1 10227.092,E2 10227.092} C_VEL
LIN {X 0,Y 339.647,Z 523.544,A -85,B 0,C 180,E1 10223.301,E2 10223.301} C_VEL
LIN {X 0,Y 343.599,Z 529.134,A -85,B 0,C 180,E1 10220.626,E2 10220.626} C_VEL
LIN {X 0,Y 348.836,Z 536.666,A -85,B 0,C 180,E1 10217.544,E2 10217.544} C_VEL
LIN {X 0,Y 356.532,Z 548.441,A -85,B 0,C 180,E1 10213.652,E2 10213.652} C_VEL
LIN {X 0,Y 357.449,Z 550.182,A -85,B 0,C 180,E1 10213.208,E2 10213.208} C_VEL
LIN {X 0,Y 342.114,Z 719.464,A -85,B 0,C 180,E1 10209.821,E2 10209.821} C_VEL
LIN {X 0,Y 338.491,Z 743.163,A -85,B 0,C 180,E1 10209.185,E2 10209.185} C_VEL
LIN {X 0,Y 334.022,Z 765.208,A -85,B 0,C 180,E1 10208.39,E2 10208.39} C_VEL
LIN {X 0,Y 328.265,Z 787.16,A -85,B 0,C 180,E1 10207.346,E2 10207.346} C_VEL
LIN {X 0,Y 321.533,Z 808.837,A -85,B 0,C 180,E1 10206.048,E2 10206.048} C_VEL
LIN {X 0,Y 314.358,Z 828.454,A -85,B 0,C 180,E1 10204.585,E2 10204.585} C_VEL
LIN {X 0,Y 305.637,Z 849.417,A -85,B 0,C 180,E1 10202.66,E2 10202.66} C_VEL
LIN {X 0,Y 297.534,Z 866.81,A -85,B 0,C 180,E1 10200.709,E2 10200.709} C_VEL
LIN {X 0,Y 287.977,Z 885.366,A -85,B 0,C 180,E1 10198.169,E2 10198.169} C_VEL
LIN {X 0,Y 278.954,Z 901.534,A -85,B 0,C 180,E1 10195.467,E2 10195.467} C_VEL
LIN {X 0,Y 269.466,Z 917.268,A -85,B 0,C 180,E1 10192.231,E2 10192.231} C_VEL
LIN {X 0,Y 260.346,Z 931.806,A -85,B 0,C 180,E1 10188.58,E2 10188.58} C_VEL
LIN {X 0,Y 252.113,Z 944.246,A -85,B 0,C 180,E1 10184.696,E2 10184.696} C_VEL
LIN {X 0,Y 244.241,Z 956.157,A -85,B 0,C 180,E1 10180.131,E2 10180.131} C_VEL
LIN {X 0,Y 237.945,Z 965.725,A -85,B 0,C 180,E1 10175.539,E2 10175.539} C_VEL
LIN {X 0,Y 232.239,Z 974.935,A -85,B 0,C 180,E1 10169.993,E2 10169.993} C_VEL
LIN {X 0,Y 228.617,Z 981.429,A -85,B 0,C 180,E1 10164.974,E2 10164.974} C_VEL
LIN {X 0,Y 225.906,Z 987.267,A -85,B 0,C 180,E1 10159.021,E2 10159.021} C_VEL
LIN {X 0,Y 224.672,Z 990.824,A -85,B 0,C 180,E1 10153.976,E2 10153.976} C_VEL
LIN {X 0,Y 224.132,Z 993.362,A -85,B 0,C 180,E1 10148.535,E2 10148.535} C_VEL
LIN {X 0,Y 224.013,Z 994.404,A -85,B 0,C 180,E1 10143.769,E2 10143.769} C_VEL
LIN {X 0,Y 224.036,Z 994.499,A -85,B 0,C 180,E1 10139.41,E2 10139.41} C_VEL
LIN {X 0,Y 224.207,Z 993.649,A -85,B 0,C 180,E1 10134.56,E2 10134.56} C_VEL
LIN {X 0,Y 224.943,Z 991.263,A -85,B 0,C 180,E1 10128.855,E2 10128.855} C_VEL
LIN {X 0,Y 226.541,Z 987.719,A -85,B 0,C 180,E1 10123.515,E2 10123.515} C_VEL
LIN {X 0,Y 229.969,Z 981.808,A -85,B 0,C 180,E1 10117.274,E2 10117.274} C_VEL
LIN {X 0,Y 234.569,Z 975.054,A -85,B 0,C 180,E1 10111.909,E2 10111.909} C_VEL
LIN {X 0,Y 240.856,Z 966.416,A -85,B 0,C 180,E1 10106.638,E2 10106.638} C_VEL
LIN {X 0,Y 248.624,Z 956.299,A -85,B 0,C 180,E1 10101.71,E2 10101.71} C_VEL
LIN {X 0,Y 257.552,Z 944.58,A -85,B 0,C 180,E1 10097.236,E2 10097.236} C_VEL
LIN {X 0,Y 268.179,Z 930.453,A -85,B 0,C 180,E1 10092.927,E2 10092.927} C_VEL
LIN {X 0,Y 273.481,Z 923.223,A -85,B 0,C 180,E1 10091.067,E2 10091.067} C_VEL
LIN {X 0,Y 276.07,Z 918.804,A -85,B 0,C 180,E1 10089.849,E2 10089.849} C_VEL
LIN {X 0,Y 280.637,Z 908.247,A -85,B 0,C 180,E1 10086.451,E2 10086.451} C_VEL
LIN {X 0,Y 283.468,Z 903.423,A -85,B 0,C 180,E1 10085.362,E2 10085.362} C_VEL
LIN {X 0,Y 294.182,Z 887.377,A -85,B 0,C 180,E1 10082.728,E2 10082.728} C_VEL
LIN {X 0,Y 305.926,Z 868.134,A -85,B 0,C 180,E1 10080.188,E2 10080.188} C_VEL
LIN {X 0,Y 316.368,Z 849.293,A -85,B 0,C 180,E1 10078.19,E2 10078.19} C_VEL
LIN {X 0,Y 326.113,Z 829.207,A -85,B 0,C 180,E1 10076.485,E2 10076.485} C_VEL
LIN {X 0,Y 335.637,Z 806.815,A -85,B 0,C 180,E1 10074.968,E2 10074.968} C_VEL
LIN {X 0,Y 342.919,Z 786.648,A -85,B 0,C 180,E1 10073.887,E2 10073.887} C_VEL
LIN {X 0,Y 349.797,Z 763.621,A -85,B 0,C 180,E1 10072.92,E2 10072.92} C_VEL
LIN {X 0,Y 354.69,Z 743.16,A -85,B 0,C 180,E1 10072.265,E2 10072.265} C_VEL
LIN {X 0,Y 358.807,Z 719.505,A -85,B 0,C 180,E1 10071.696,E2 10071.696} C_VEL
LIN {X 0,Y 377.785,Z 567.664,A -85,B 0,C 180,E1 10068.726,E2 10068.726} C_VEL
LIN {X 0,Y 377.384,Z 566.198,A -85,B 0,C 180,E1 10066.049,E2 10066.049} C_VEL
LIN {X 0,Y 377.797,Z 567.924,A -85,B 0,C 180,E1 10063.642,E2 10063.642} C_VEL
LIN {X 0,Y 357.657,Z 728.754,A -85,B 0,C 180,E1 10060.492,E2 10060.492} C_VEL
LIN {X 0,Y 352.969,Z 752.796,A -85,B 0,C 180,E1 10059.914,E2 10059.914} C_VEL
LIN {X 0,Y 347.059,Z 775.828,A -85,B 0,C 180,E1 10059.215,E2 10059.215} C_VEL
LIN {X 0,Y 340.826,Z 795.277,A -85,B 0,C 180,E1 10058.437,E2 10058.437} C_VEL
LIN {X 0,Y 332.694,Z 817.122,A -85,B 0,C 180,E1 10057.323,E2 10057.323} C_VEL
LIN {X 0,Y 324.33,Z 836.289,A -85,B 0,C 180,E1 10056.081,E2 10056.081} C_VEL
LIN {X 0,Y 314.168,Z 857.176,A -85,B 0,C 180,E1 10054.394,E2 10054.394} C_VEL
LIN {X 0,Y 303.487,Z 876.638,A -85,B 0,C 180,E1 10052.412,E2 10052.412} C_VEL
LIN {X 0,Y 291.758,Z 896.106,A -85,B 0,C 180,E1 10049.927,E2 10049.927} C_VEL
LIN {X 0,Y 281.334,Z 912.17,A -85,B 0,C 180,E1 10047.391,E2 10047.391} C_VEL
LIN {X 0,Y 269.925,Z 928.601,A -85,B 0,C 180,E1 10044.179,E2 10044.179} C_VEL
LIN {X 0,Y 258.516,Z 944.385,A -85,B 0,C 180,E1 10040.332,E2 10040.332} C_VEL
LIN {X 0,Y 248.281,Z 957.968,A -85,B 0,C 180,E1 10036.133,E2 10036.133} C_VEL
LIN {X 0,Y 238.205,Z 971.372,A -85,B 0,C 180,E1 10030.913,E2 10030.913} C_VEL
LIN {X 0,Y 230.689,Z 981.735,A -85,B 0,C 180,E1 10025.819,E2 10025.819} C_VEL
LIN {X 0,Y 224.573,Z 990.675,A -85,B 0,C 180,E1 10020.213,E2 10020.213} C_VEL
LIN {X 0,Y 220.258,Z 998.024,A -85,B 0,C 180,E1 10014.407,E2 10014.407} C_VEL
LIN {X 0,Y 217.606,Z 1003.568,A -85,B 0,C 180,E1 10008.492,E2 10008.492} C_VEL
LIN {X 0,Y 216.315,Z 1007.69,A -85,B 0,C 180,E1 10002.555,E2 10002.555} C_VEL
LIN {X 0,Y 215.989,Z 1009.939,A -85,B 0,C 180,E1 9997.188,E2 9997.188} C_VEL
LIN {X 0,Y 216.005,Z 1010.891,A -85,B 0,C 180,E1 9992.661,E2 9992.661} C_VEL
LIN {X 0,Y 216.026,Z 1010.938,A -85,B 0,C 180,E1 9988.417,E2 9988.417} C_VEL
LIN {X 0,Y 216.008,Z 1010.008,A -85,B 0,C 180,E1 9983.63,E2 9983.63} C_VEL
LIN {X 0,Y 216.23,Z 1007.699,A -85,B 0,C 180,E1 9978.269,E2 9978.269} C_VEL
LIN {X 0,Y 217.116,Z 1004.212,A -85,B 0,C 180,E1 9973.144,E2 9973.144} C_VEL
LIN {X 0,Y 219.215,Z 999.014,A -85,B 0,C 180,E1 9967.482,E2 9967.482} C_VEL
LIN {X 0,Y 222.926,Z 991.715,A -85,B 0,C 180,E1 9961.623,E2 9961.623} C_VEL
LIN {X 0,Y 228.088,Z 983.144,A -85,B 0,C 180,E1 9956.181,E2 9956.181} C_VEL
LIN {X 0,Y 234.503,Z 973.131,A -85,B 0,C 180,E1 9951.199,E2 9951.199} C_VEL
LIN {X 0,Y 242.812,Z 960.696,A -85,B 0,C 180,E1 9946.24,E2 9946.24} C_VEL
LIN {X 0,Y 251.148,Z 948.187,A -85,B 0,C 180,E1 9942.239,E2 9942.239} C_VEL
LIN {X 0,Y 261.098,Z 932.843,A -85,B 0,C 180,E1 9938.29,E2 9938.29} C_VEL
LIN {X 0,Y 270.913,Z 917.024,A -85,B 0,C 180,E1 9934.996,E2 9934.996} C_VEL
LIN {X 0,Y 280.873,Z 899.654,A -85,B 0,C 180,E1 9932.103,E2 9932.103} C_VEL
LIN {X 0,Y 291.014,Z 880.604,A -85,B 0,C 180,E1 9929.529,E2 9929.529} C_VEL
LIN {X 0,Y 299.86,Z 862.251,A -85,B 0,C 180,E1 9927.524,E2 9927.524} C_VEL
LIN {X 0,Y 308.867,Z 841.297,A -85,B 0,C 180,E1 9925.676,E2 9925.676} C_VEL
LIN {X 0,Y 316.755,Z 820.476,A -85,B 0,C 180,E1 9924.201,E2 9924.201} C_VEL
LIN {X 0,Y 323.647,Z 798.952,A -85,B 0,C 180,E1 9923.001,E2 9923.001} C_VEL
LIN {X 0,Y 329.817,Z 776.119,A -85,B 0,C 180,E1 9922.006,E2 9922.006} C_VEL
LIN {X 0,Y 334.593,Z 753.616,A -85,B 0,C 180,E1 9921.282,E2 9921.282} C_VEL
LIN {X 0,Y 338.349,Z 728.472,A -85,B 0,C 180,E1 9920.655,E2 9920.655} C_VEL
LIN {X 0,Y 354.271,Z 556.249,A -85,B 0,C 180,E1 9917.216,E2 9917.216} C_VEL
LIN {X 0,Y 349.262,Z 547.643,A -85,B 0,C 180,E1 9914.633,E2 9914.633} C_VEL
LIN {X 0,Y 343.245,Z 538.602,A -85,B 0,C 180,E1 9911.169,E2 9911.169} C_VEL
LIN {X 0,Y 339.652,Z 533.496,A -85,B 0,C 180,E1 9908.805,E2 9908.805} C_VEL
LIN {X 0,Y 336.643,Z 529.156,A -85,B 0,C 180,E1 9906.565,E2 9906.565} C_VEL
LIN {X 0,Y 333.373,Z 524.55,A -85,B 0,C 180,E1 9903.783,E2 9903.783} C_VEL
LIN {X 0,Y 330.272,Z 520.157,A -85,B 0,C 180,E1 9900.606,E2 9900.606} C_VEL
LIN {X 0,Y 326.737,Z 515.574,A -85,B 0,C 180,E1 9895.788,E2 9895.788} C_VEL
LIN {X 0,Y 326.138,Z 514.113,A -85,B 0,C 180,E1 9894.546,E2 9894.546} C_VEL
LIN {X 0,Y 323.813,Z 512.355,A -85,B 0,C 180,E1 9887.517,E2 9887.517} C_VEL
LIN {X 0,Y 323.932,Z 512.459,A -85,B 0,C 180,E1 9882.948,E2 9882.948} C_VEL
LIN {X 0,Y 326.319,Z 514.385,A -85,B 0,C 180,E1 9876.334,E2 9876.334} C_VEL
LIN {X 0,Y 328.742,Z 518.544,A -85,B 0,C 180,E1 9872.463,E2 9872.463} C_VEL
LIN {X 0,Y 330.377,Z 520.291,A -85,B 0,C 180,E1 9870.541,E2 9870.541} C_VEL
LIN {X 0,Y 334.339,Z 525.897,A -85,B 0,C 180,E1 9866.614,E2 9866.614} C_VEL
LIN {X 0,Y 338.051,Z 531.154,A -85,B 0,C 180,E1 9863.627,E2 9863.627} C_VEL
LIN {X 0,Y 341.871,Z 536.653,A -85,B 0,C 180,E1 9860.983,E2 9860.983} C_VEL
LIN {X 0,Y 346.941,Z 544.109,A -85,B 0,C 180,E1 9857.928,E2 9857.928} C_VEL
LIN {X 0,Y 353.901,Z 554.946,A -85,B 0,C 180,E1 9854.309,E2 9854.309} C_VEL
LIN {X 0,Y 338.558,Z 719.626,A -85,B 0,C 180,E1 9851.029,E2 9851.029} C_VEL
LIN {X 0,Y 334.832,Z 743.47,A -85,B 0,C 180,E1 9850.396,E2 9850.396} C_VEL
LIN {X 0,Y 330.168,Z 765.879,A -85,B 0,C 180,E1 9849.594,E2 9849.594} C_VEL
LIN {X 0,Y 324.492,Z 787.079,A -85,B 0,C 180,E1 9848.598,E2 9848.598} C_VEL
LIN {X 0,Y 317.541,Z 809.023,A -85,B 0,C 180,E1 9847.302,E2 9847.302} C_VEL
LIN {X 0,Y 310.366,Z 828.229,A -85,B 0,C 180,E1 9845.888,E2 9845.888} C_VEL
LIN {X 0,Y 301.559,Z 848.961,A -85,B 0,C 180,E1 9844.012,E2 9844.012} C_VEL
LIN {X 0,Y 293.047,Z 866.743,A -85,B 0,C 180,E1 9842.035,E2 9842.035} C_VEL
LIN {X 0,Y 282.883,Z 885.908,A -85,B 0,C 180,E1 9839.418,E2 9839.418} C_VEL
LIN {X 0,Y 273.564,Z 902.098,A -85,B 0,C 180,E1 9836.707,E2 9836.707} C_VEL
LIN {X 0,Y 263.728,Z 917.824,A -85,B 0,C 180,E1 9833.45,E2 9833.45} C_VEL
LIN {X 0,Y 254.243,Z 932.323,A -85,B 0,C 180,E1 9829.76,E2 9829.76} C_VEL
LIN {X 0,Y 245.238,Z 945.372,A -85,B 0,C 180,E1 9825.602,E2 9825.602} C_VEL
LIN {X 0,Y 236.695,Z 957.657,A -85,B 0,C 180,E1 9820.704,E2 9820.704} C_VEL
LIN {X 0,Y 230.207,Z 967.108,A -85,B 0,C 180,E1 9815.975,E2 9815.975} C_VEL
LIN {X 0,Y 224.541,Z 975.725,A -85,B 0,C 180,E1 9810.502,E2 9810.502} C_VEL
LIN {X 0,Y 220.614,Z 982.463,A -85,B 0,C 180,E1 9805.052,E2 9805.052} C_VEL
LIN {X 0,Y 217.917,Z 987.922,A -85,B 0,C 180,E1 9799.084,E2 9799.084} C_VEL
LIN {X 0,Y 216.591,Z 991.699,A -85,B 0,C 180,E1 9793.361,E2 9793.361} C_VEL
LIN {X 0,Y 216.103,Z 993.918,A -85,B 0,C 180,E1 9787.696,E2 9787.696} C_VEL
LIN {X 0,Y 216.021,Z 994.75,A -85,B 0,C 180,E1 9783.294,E2 9783.294} C_VEL
LIN {X 0,Y 216.068,Z 994.775,A -85,B 0,C 180,E1 9778.775,E2 9778.775} C_VEL
LIN {X 0,Y 216.328,Z 993.658,A -85,B 0,C 180,E1 9773.094,E2 9773.094} C_VEL
LIN {X 0,Y 217.195,Z 991.297,A -85,B 0,C 180,E1 9767.761,E2 9767.761} C_VEL
LIN {X 0,Y 219.124,Z 987.604,A -85,B 0,C 180,E1 9762.127,E2 9762.127} C_VEL
LIN {X 0,Y 222.749,Z 981.935,A -85,B 0,C 180,E1 9756.092,E2 9756.092} C_VEL
LIN {X 0,Y 228.118,Z 974.739,A -85,B 0,C 180,E1 9750.27,E2 9750.27} C_VEL
LIN {X 0,Y 234.996,Z 965.965,A -85,B 0,C 180,E1 9744.913,E2 9744.913} C_VEL
LIN {X 0,Y 243.966,Z 954.974,A -85,B 0,C 180,E1 9739.638,E2 9739.638} C_VEL
LIN {X 0,Y 253.152,Z 943.658,A -85,B 0,C 180,E1 9735.346,E2 9735.346} C_VEL
LIN {X 0,Y 264.018,Z 929.875,A -85,B 0,C 180,E1 9731.207,E2 9731.207} C_VEL
LIN {X 0,Y 274.935,Z 915.476,A -85,B 0,C 180,E1 9727.734,E2 9727.734} C_VEL
LIN {X 0,Y 283.468,Z 903.423,A -85,B 0,C 180,E1 9725.362,E2 9725.362} C_VEL
LIN {X 0,Y 286.378,Z 898.527,A -85,B 0,C 180,E1 9724.303,E2 9724.303} C_VEL
LIN {X 0,Y 291.982,Z 886.729,A -85,B 0,C 180,E1 9721.269,E2 9721.269} C_VEL
LIN {X 0,Y 295.04,Z 881.417,A -85,B 0,C 180,E1 9720.344,E2 9720.344} C_VEL
LIN {X 0,Y 306.282,Z 863.183,A -85,B 0,C 180,E1 9718.13,E2 9718.13} C_VEL
LIN {X 0,Y 316.636,Z 844.312,A -85,B 0,C 180,E1 9716.29,E2 9716.29} C_VEL
LIN {X 0,Y 326.374,Z 824.543,A -85,B 0,C 180,E1 9714.727,E2 9714.727} C_VEL
LIN {X 0,Y 335.184,Z 803.614,A -85,B 0,C 180,E1 9713.411,E2 9713.411} C_VEL
LIN {X 0,Y 343.045,Z 781.783,A -85,B 0,C 180,E1 9712.322,E2 9712.322} C_VEL
LIN {X 0,Y 349.403,Z 760.133,A -85,B 0,C 180,E1 9711.483,E2 9711.483} C_VEL
LIN {X 0,Y 354.941,Z 735.759,A -85,B 0,C 180,E1 9710.781,E2 9710.781} C_VEL
LIN {X 0,Y 358.801,Z 711.773,A -85,B 0,C 180,E1 9710.264,E2 9710.264} C_VEL
LIN {X 0,Y 376.386,Z 574.915,A -85,B 0,C 180,E1 9707.653,E2 9707.653} C_VEL
LIN {X 0,Y 376.285,Z 574.175,A -85,B 0,C 180,E1 9706.008,E2 9706.008} C_VEL
LIN {X 0,Y 376.38,Z 575.043,A -85,B 0,C 180,E1 9704.728,E2 9704.728} C_VEL
LIN {X 0,Y 356.533,Z 728.223,A -85,B 0,C 180,E1 9701.779,E2 9701.779} C_VEL
LIN {X 0,Y 351.731,Z 752.309,A -85,B 0,C 180,E1 9701.218,E2 9701.218} C_VEL
LIN {X 0,Y 345.706,Z 775.218,A -85,B 0,C 180,E1 9700.547,E2 9700.547} C_VEL
LIN {X 0,Y 339.335,Z 794.573,A -85,B 0,C 180,E1 9699.804,E2 9699.804} C_VEL
LIN {X 0,Y 331.059,Z 816.29,A -85,B 0,C 180,E1 9698.738,E2 9698.738} C_VEL
LIN {X 0,Y 322.042,Z 836.325,A -85,B 0,C 180,E1 9697.476,E2 9697.476} C_VEL
LIN {X 0,Y 311.349,Z 857.495,A -85,B 0,C 180,E1 9695.796,E2 9695.796} C_VEL
LIN {X 0,Y 300.621,Z 876.376,A -85,B 0,C 180,E1 9693.907,E2 9693.907} C_VEL
LIN {X 0,Y 288.508,Z 895.737,A -85,B 0,C 180,E1 9691.475,E2 9691.475} C_VEL
LIN {X 0,Y 277.03,Z 912.711,A -85,B 0,C 180,E1 9688.81,E2 9688.81} C_VEL
LIN {X 0,Y 265.275,Z 928.822,A -85,B 0,C 180,E1 9685.641,E2 9685.641} C_VEL
LIN {X 0,Y 253.875,Z 943.843,A -85,B 0,C 180,E1 9681.977,E2 9681.977} C_VEL
LIN {X 0,Y 243.085,Z 957.402,A -85,B 0,C 180,E1 9677.772,E2 9677.772} C_VEL
LIN {X 0,Y 232.781,Z 970.302,A -85,B 0,C 180,E1 9672.737,E2 9672.737} C_VEL
LIN {X 0,Y 224.654,Z 980.708,A -85,B 0,C 180,E1 9667.579,E2 9667.579} C_VEL
LIN {X 0,Y 217.67,Z 990.145,A -85,B 0,C 180,E1 9661.586,E2 9661.586} C_VEL
LIN {X 0,Y 212.899,Z 997.522,A -85,B 0,C 180,E1 9655.607,E2 9655.607} C_VEL
LIN {X 0,Y 209.874,Z 1003.186,A -85,B 0,C 180,E1 9649.392,E2 9649.392} C_VEL
LIN {X 0,Y 208.417,Z 1007.271,A -85,B 0,C 180,E1 9643.321,E2 9643.321} C_VEL
LIN {X 0,Y 208.004,Z 1009.578,A -85,B 0,C 180,E1 9637.743,E2 9637.743} C_VEL
LIN {X 0,Y 208.002,Z 1010.566,A -85,B 0,C 180,E1 9633.039,E2 9633.039} C_VEL
LIN {X 0,Y 208.031,Z 1010.643,A -85,B 0,C 180,E1 9628.569,E2 9628.569} C_VEL
LIN {X 0,Y 208.011,Z 1009.752,A -85,B 0,C 180,E1 9623.661,E2 9623.661} C_VEL
LIN {X 0,Y 208.245,Z 1007.5,A -85,B 0,C 180,E1 9618.094,E2 9618.094} C_VEL
LIN {X 0,Y 209.276,Z 1003.823,A -85,B 0,C 180,E1 9612.492,E2 9612.492} C_VEL
LIN {X 0,Y 211.723,Z 998.304,A -85,B 0,C 180,E1 9606.344,E2 9606.344} C_VEL
LIN {X 0,Y 215.606,Z 991.253,A -85,B 0,C 180,E1 9600.567,E2 9600.567} C_VEL
LIN {X 0,Y 221.461,Z 982.133,A -85,B 0,C 180,E1 9594.708,E2 9594.708} C_VEL
LIN {X 0,Y 227.999,Z 972.554,A -85,B 0,C 180,E1 9589.873,E2 9589.873} C_VEL
LIN {X 0,Y 236.783,Z 960.049,A -85,B 0,C 180,E1 9584.826,E2 9584.826} C_VEL
LIN {X 0,Y 245.556,Z 947.48,A -85,B 0,C 180,E1 9580.782,E2 9580.782} C_VEL
LIN {X 0,Y 255.379,Z 932.891,A -85,B 0,C 180,E1 9577.008,E2 9577.008} C_VEL
LIN {X 0,Y 265.544,Z 917.103,A -85,B 0,C 180,E1 9573.696,E2 9573.696} C_VEL
LIN {X 0,Y 275.833,Z 899.797,A -85,B 0,C 180,E1 9570.801,E2 9570.801} C_VEL
LIN {X 0,Y 286.07,Z 881.184,A -85,B 0,C 180,E1 9568.281,E2 9568.281} C_VEL
LIN {X 0,Y 295.356,Z 862.43,A -85,B 0,C 180,E1 9566.239,E2 9566.239} C_VEL
LIN {X 0,Y 304.591,Z 841.57,A -85,B 0,C 180,E1 9564.408,E2 9564.408} C_VEL
LIN {X 0,Y 312.661,Z 820.816,A -85,B 0,C 180,E1 9562.948,E2 9562.948} C_VEL
LIN {X 0,Y 319.706,Z 799.466,A -85,B 0,C 180,E1 9561.764,E2 9561.764} C_VEL
LIN {X 0,Y 326.003,Z 776.903,A -85,B 0,C 180,E1 9560.784,E2 9560.784} C_VEL
LIN {X 0,Y 331.007,Z 753.875,A -85,B 0,C 180,E1 9560.051,E2 9560.051} C_VEL
LIN {X 0,Y 334.909,Z 728.455,A -85,B 0,C 180,E1 9559.422,E2 9559.422} C_VEL
LIN {X 0,Y 350.783,Z 561.061,A -85,B 0,C 180,E1 9556.097,E2 9556.097} C_VEL
LIN {X 0,Y 346.46,Z 553.775,A -85,B 0,C 180,E1 9553.773,E2 9553.773} C_VEL
LIN {X 0,Y 340.981,Z 545.379,A -85,B 0,C 180,E1 9550.474,E2 9550.474} C_VEL
LIN {X 0,Y 337.72,Z 540.665,A -85,B 0,C 180,E1 9548.255,E2 9548.255} C_VEL
LIN {X 0,Y 334.993,Z 536.663,A -85,B 0,C 180,E1 9546.168,E2 9546.168} C_VEL
LIN {X 0,Y 331.886,Z 532.207,A -85,B 0,C 180,E1 9543.454,E2 9543.454} C_VEL
LIN {X 0,Y 328.501,Z 527.327,A -85,B 0,C 180,E1 9539.825,E2 9539.825} C_VEL
LIN {X 0,Y 325.618,Z 523.628,A -85,B 0,C 180,E1 9535.773,E2 9535.773} C_VEL
LIN {X 0,Y 324.944,Z 521.987,A -85,B 0,C 180,E1 9534.349,E2 9534.349} C_VEL
LIN {X 0,Y 322.701,Z 520.258,A -85,B 0,C 180,E1 9527.291,E2 9527.291} C_VEL
LIN {X 0,Y 322.876,Z 520.438,A -85,B 0,C 180,E1 9522.705,E2 9522.705} C_VEL
LIN {X 0,Y 325.115,Z 522.242,A -85,B 0,C 180,E1 9516.53,E2 9516.53} C_VEL
LIN {X 0,Y 327.574,Z 526.456,A -85,B 0,C 180,E1 9512.554,E2 9512.554} C_VEL
LIN {X 0,Y 329.023,Z 528.038,A -85,B 0,C 180,E1 9510.807,E2 9510.807} C_VEL
LIN {X 0,Y 332.866,Z 533.564,A -85,B 0,C 180,E1 9506.922,E2 9506.922} C_VEL
LIN {X 0,Y 336.539,Z 538.882,A -85,B 0,C 180,E1 9503.9,E2 9503.9} C_VEL
LIN {X 0,Y 340.225,Z 544.275,A -85,B 0,C 180,E1 9501.3,E2 9501.3} C_VEL
LIN {X 0,Y 345.138,Z 551.679,A -85,B 0,C 180,E1 9498.272,E2 9498.272} C_VEL
LIN {X 0,Y 350.403,Z 560.176,A -85,B 0,C 180,E1 9495.415,E2 9495.415} C_VEL
LIN {X 0,Y 335.131,Z 719.907,A -85,B 0,C 180,E1 9492.258,E2 9492.258} C_VEL
LIN {X 0,Y 331.348,Z 743.641,A -85,B 0,C 180,E1 9491.636,E2 9491.636} C_VEL
LIN {X 0,Y 326.647,Z 765.807,A -85,B 0,C 180,E1 9490.856,E2 9490.856} C_VEL
LIN {X 0,Y 320.656,Z 787.676,A -85,B 0,C 180,E1 9489.841,E2 9489.841} C_VEL
LIN {X 0,Y 313.536,Z 809.559,A -85,B 0,C 180,E1 9488.559,E2 9488.559} C_VEL
LIN {X 0,Y 306.18,Z 828.748,A -85,B 0,C 180,E1 9487.158,E2 9487.158} C_VEL
LIN {X 0,Y 296.898,Z 849.988,A -85,B 0,C 180,E1 9485.242,E2 9485.242} C_VEL
LIN {X 0,Y 288.073,Z 867.925,A -85,B 0,C 180,E1 9483.248,E2 9483.248} C_VEL
LIN {X 0,Y 277.928,Z 886.441,A -85,B 0,C 180,E1 9480.712,E2 9480.712} C_VEL
LIN {X 0,Y 268.3,Z 902.622,A -85,B 0,C 180,E1 9477.997,E2 9477.997} C_VEL
LIN {X 0,Y 258.108,Z 918.325,A -85,B 0,C 180,E1 9474.723,E2 9474.723} C_VEL
LIN {X 0,Y 248.248,Z 932.826,A -85,B 0,C 180,E1 9470.997,E2 9470.997} C_VEL
LIN {X 0,Y 239.311,Z 945.258,A -85,B 0,C 180,E1 9466.997,E2 9466.997} C_VEL
LIN {X 0,Y 230.289,Z 957.622,A -85,B 0,C 180,E1 9462.021,E2 9462.021} C_VEL
LIN {X 0,Y 223.397,Z 967.123,A -85,B 0,C 180,E1 9457.191,E2 9457.191} C_VEL
LIN {X 0,Y 217.337,Z 975.818,A -85,B 0,C 180,E1 9451.574,E2 9451.574} C_VEL
LIN {X 0,Y 213.252,Z 982.284,A -85,B 0,C 180,E1 9446.228,E2 9446.228} C_VEL
LIN {X 0,Y 210.165,Z 988.045,A -85,B 0,C 180,E1 9439.854,E2 9439.854} C_VEL
LIN {X 0,Y 208.709,Z 991.733,A -85,B 0,C 180,E1 9434.145,E2 9434.145} C_VEL
LIN {X 0,Y 208.129,Z 994.098,A -85,B 0,C 180,E1 9428.282,E2 9428.282} C_VEL
LIN {X 0,Y 208.025,Z 995.031,A -85,B 0,C 180,E1 9423.441,E2 9423.441} C_VEL
LIN {X 0,Y 208.075,Z 995.096,A -85,B 0,C 180,E1 9418.8,E2 9418.8} C_VEL
LIN {X 0,Y 208.335,Z 994.13,A -85,B 0,C 180,E1 9413.128,E2 9413.128} C_VEL
LIN {X 0,Y 209.311,Z 991.712,A -85,B 0,C 180,E1 9407.278,E2 9407.278} C_VEL
LIN {X 0,Y 211.34,Z 988.182,A -85,B 0,C 180,E1 9401.616,E2 9401.616} C_VEL
LIN {X 0,Y 215.378,Z 982.415,A -85,B 0,C 180,E1 9395.146,E2 9395.146} C_VEL
LIN {X 0,Y 221.097,Z 975.333,A -85,B 0,C 180,E1 9389.203,E2 9389.203} C_VEL
LIN {X 0,Y 228.622,Z 966.392,A -85,B 0,C 180,E1 9383.576,E2 9383.576} C_VEL
LIN {X 0,Y 238.007,Z 955.619,A -85,B 0,C 180,E1 9378.285,E2 9378.285} C_VEL
LIN {X 0,Y 248.168,Z 943.799,A -85,B 0,C 180,E1 9373.752,E2 9373.752} C_VEL
LIN {X 0,Y 259.618,Z 929.965,A -85,B 0,C 180,E1 9369.598,E2 9369.598} C_VEL
LIN {X 0,Y 271.035,Z 915.56,A -85,B 0,C 180,E1 9366.142,E2 9366.142} C_VEL
LIN {X 0,Y 282.414,Z 900.01,A -85,B 0,C 180,E1 9363.179,E2 9363.179} C_VEL
LIN {X 0,Y 294.823,Z 881.76,A -85,B 0,C 180,E1 9360.389,E2 9360.389} C_VEL
LIN {X 0,Y 295.04,Z 881.417,A -85,B 0,C 180,E1 9360.344,E2 9360.344} C_VEL
LIN {X 0,Y 298.147,Z 876.046,A -85,B 0,C 180,E1 9359.45,E2 9359.45} C_VEL
LIN {X 0,Y 304.814,Z 862.297,A -85,B 0,C 180,E1 9356.658,E2 9356.658} C_VEL
LIN {X 0,Y 307.516,Z 857.262,A -85,B 0,C 180,E1 9356.009,E2 9356.009} C_VEL
LIN {X 0,Y 317.944,Z 838.361,A -85,B 0,C 180,E1 9354.325,E2 9354.325} C_VEL
LIN {X 0,Y 327.477,Z 818.471,A -85,B 0,C 180,E1 9352.908,E2 9352.908} C_VEL
LIN {X 0,Y 336.126,Z 797.956,A -85,B 0,C 180,E1 9351.729,E2 9351.729} C_VEL
LIN {X 0,Y 343.406,Z 776.998,A -85,B 0,C 180,E1 9350.779,E2 9350.779} C_VEL
LIN {X 0,Y 349.974,Z 754.169,A -85,B 0,C 180,E1 9349.976,E2 9349.976} C_VEL
LIN {X 0,Y 354.762,Z 732.12,A -85,B 0,C 180,E1 9349.402,E2 9349.402} C_VEL
LIN {X 0,Y 359.504,Z 700.158,A -85,B 0,C 180,E1 9348.763,E2 9348.763} C_VEL
LIN {X 0,Y 375.203,Z 582.21,A -85,B 0,C 180,E1 9346.556,E2 9346.556} C_VEL
LIN {X 0,Y 375.192,Z 582.253,A -85,B 0,C 180,E1 9345.823,E2 9345.823} C_VEL
LIN {X 0,Y 355.715,Z 727.641,A -85,B 0,C 180,E1 9343.078,E2 9343.078} C_VEL
LIN {X 0,Y 350.881,Z 751.44,A -85,B 0,C 180,E1 9342.543,E2 9342.543} C_VEL
LIN {X 0,Y 344.774,Z 774.244,A -85,B 0,C 180,E1 9341.904,E2 9341.904} C_VEL
LIN {X 0,Y 338.056,Z 794.178,A -85,B 0,C 180,E1 9341.175,E2 9341.175} C_VEL
LIN {X 0,Y 329.558,Z 815.863,A -85,B 0,C 180,E1 9340.148,E2 9340.148} C_VEL
LIN {X 0,Y 319.554,Z 837.411,A -85,B 0,C 180,E1 9338.824,E2 9338.824} C_VEL
LIN {X 0,Y 308.2,Z 858.879,A -85,B 0,C 180,E1 9337.133,E2 9337.133} C_VEL
LIN {X 0,Y 297.209,Z 877.517,A -85,B 0,C 180,E1 9335.284,E2 9335.284} C_VEL
LIN {X 0,Y 285.117,Z 896.007,A -85,B 0,C 180,E1 9332.975,E2 9332.975} C_VEL
LIN {X 0,Y 272.911,Z 913.342,A -85,B 0,C 180,E1 9330.27,E2 9330.27} C_VEL
LIN {X 0,Y 260.735,Z 929.226,A -85,B 0,C 180,E1 9327.129,E2 9327.129} C_VEL
LIN {X 0,Y 248.865,Z 944.054,A -85,B 0,C 180,E1 9323.478,E2 9323.478} C_VEL
LIN {X 0,Y 237.691,Z 957.374,A -85,B 0,C 180,E1 9319.308,E2 9319.308} C_VEL
LIN {X 0,Y 226.73,Z 970.282,A -85,B 0,C 180,E1 9314.176,E2 9314.176} C_VEL
LIN {X 0,Y 217.772,Z 981.052,A -85,B 0,C 180,E1 9308.693,E2 9308.693} C_VEL
LIN {X 0,Y 210.608,Z 990.005,A -85,B 0,C 180,E1 9302.775,E2 9302.775} C_VEL
LIN {X 0,Y 205.254,Z 997.609,A -85,B 0,C 180,E1 9296.324,E2 9296.324} C_VEL
LIN {X 0,Y 202.043,Z 1003.104,A -85,B 0,C 180,E1 9289.974,E2 9289.974} C_VEL
LIN {X 0,Y 200.447,Z 1007.158,A -85,B 0,C 180,E1 9283.567,E2 9283.567} C_VEL
LIN {X 0,Y 200.007,Z 1009.375,A -85,B 0,C 180,E1 9277.766,E2 9277.766} C_VEL
LIN {X 0,Y 200.005,Z 1010.272,A -85,B 0,C 180,E1 9273.161,E2 9273.161} C_VEL
LIN {X 0,Y 200.038,Z 1010.339,A -85,B 0,C 180,E1 9268.577,E2 9268.577} C_VEL
LIN {X 0,Y 200.015,Z 1009.495,A -85,B 0,C 180,E1 9263.695,E2 9263.695} C_VEL
LIN {X 0,Y 200.261,Z 1007.299,A -85,B 0,C 180,E1 9257.905,E2 9257.905} C_VEL
LIN {X 0,Y 201.369,Z 1003.648,A -85,B 0,C 180,E1 9252.08,E2 9252.08} C_VEL
LIN {X 0,Y 203.948,Z 998.236,A -85,B 0,C 180,E1 9245.762,E2 9245.762} C_VEL
LIN {X 0,Y 208.12,Z 991.138,A -85,B 0,C 180,E1 9239.717,E2 9239.717} C_VEL
LIN {X 0,Y 214.053,Z 982.477,A -85,B 0,C 180,E1 9233.909,E2 9233.909} C_VEL
LIN {X 0,Y 221.22,Z 972.504,A -85,B 0,C 180,E1 9228.722,E2 9228.722} C_VEL
LIN {X 0,Y 230.429,Z 960.023,A -85,B 0,C 180,E1 9223.575,E2 9223.575} C_VEL
LIN {X 0,Y 239.585,Z 947.473,A -85,B 0,C 180,E1 9219.475,E2 9219.475} C_VEL
LIN {X 0,Y 249.792,Z 932.936,A -85,B 0,C 180,E1 9215.668,E2 9215.668} C_VEL
LIN {X 0,Y 260.315,Z 917.141,A -85,B 0,C 180,E1 9212.343,E2 9212.343} C_VEL
LIN {X 0,Y 270.936,Z 899.859,A -85,B 0,C 180,E1 9209.45,E2 9209.45} C_VEL
LIN {X 0,Y 281.472,Z 881.314,A -85,B 0,C 180,E1 9206.941,E2 9206.941} C_VEL
LIN {X 0,Y 291.006,Z 862.602,A -85,B 0,C 180,E1 9204.916,E2 9204.916} C_VEL
LIN {X 0,Y 300.467,Z 841.805,A -85,B 0,C 180,E1 9203.103,E2 9203.103} C_VEL
LIN {X 0,Y 308.359,Z 821.991,A -85,B 0,C 180,E1 9201.719,E2 9201.719} C_VEL
LIN {X 0,Y 315.912,Z 799.807,A -85,B 0,C 180,E1 9200.495,E2 9200.495} C_VEL
LIN {X 0,Y 322.21,Z 777.843,A -85,B 0,C 180,E1 9199.547,E2 9199.547} C_VEL
LIN {X 0,Y 327.405,Z 754.675,A -85,B 0,C 180,E1 9198.813,E2 9198.813} C_VEL
LIN {X 0,Y 331.351,Z 730.367,A -85,B 0,C 180,E1 9198.21,E2 9198.21} C_VEL
LIN {X 0,Y 347.417,Z 565.951,A -85,B 0,C 180,E1 9194.968,E2 9194.968} C_VEL
LIN {X 0,Y 342.586,Z 557.992,A -85,B 0,C 180,E1 9192.215,E2 9192.215} C_VEL
LIN {X 0,Y 337.081,Z 549.532,A -85,B 0,C 180,E1 9188.614,E2 9188.614} C_VEL
LIN {X 0,Y 333.255,Z 544.037,A -85,B 0,C 180,E1 9185.681,E2 9185.681} C_VEL
LIN {X 0,Y 330.396,Z 539.846,A -85,B 0,C 180,E1 9183.108,E2 9183.108} C_VEL
LIN {X 0,Y 327.109,Z 535.043,A -85,B 0,C 180,E1 9179.474,E2 9179.474} C_VEL
LIN {X 0,Y 324.313,Z 531.261,A -85,B 0,C 180,E1 9175.402,E2 9175.402} C_VEL
LIN {X 0,Y 323.681,Z 529.83,A -85,B 0,C 180,E1 9174.006,E2 9174.006} C_VEL
LIN {X 0,Y 321.594,Z 528.163,A -85,B 0,C 180,E1 9167.064,E2 9167.064} C_VEL
LIN {X 0,Y 321.826,Z 528.421,A -85,B 0,C 180,E1 9162.46,E2 9162.46} C_VEL
LIN {X 0,Y 323.955,Z 530.219,A -85,B 0,C 180,E1 9156.633,E2 9156.633} C_VEL
LIN {X 0,Y 326.545,Z 534.518,A -85,B 0,C 180,E1 9152.46,E2 9152.46} C_VEL
LIN {X 0,Y 327.749,Z 535.933,A -85,B 0,C 180,E1 9150.983,E2 9150.983} C_VEL
LIN {X 0,Y 331.421,Z 541.269,A -85,B 0,C 180,E1 9147.211,E2 9147.211} C_VEL
LIN {X 0,Y 335.007,Z 546.561,A -85,B 0,C 180,E1 9144.198,E2 9144.198} C_VEL
LIN {X 0,Y 338.785,Z 552.2,A -85,B 0,C 180,E1 9141.484,E2 9141.484} C_VEL
LIN {X 0,Y 343.864,Z 560.111,A -85,B 0,C 180,E1 9138.312,E2 9138.312} C_VEL
LIN {X 0,Y 347.019,Z 565.362,A -85,B 0,C 180,E1 9136.544,E2 9136.544} C_VEL
LIN {X 0,Y 331.799,Z 720.181,A -85,B 0,C 180,E1 9133.508,E2 9133.508} C_VEL
LIN {X 0,Y 327.913,Z 744.02,A -85,B 0,C 180,E1 9132.891,E2 9132.891} C_VEL
LIN {X 0,Y 323.086,Z 766.282,A -85,B 0,C 180,E1 9132.118,E2 9132.118} C_VEL
LIN {X 0,Y 316.965,Z 788.16,A -85,B 0,C 180,E1 9131.116,E2 9131.116} C_VEL
LIN {X 0,Y 309.68,Z 810.048,A -85,B 0,C 180,E1 9129.849,E2 9129.849} C_VEL
LIN {X 0,Y 302.149,Z 829.263,A -85,B 0,C 180,E1 9128.462,E2 9128.462} C_VEL
LIN {X 0,Y 292.707,Z 850.304,A -85,B 0,C 180,E1 9126.58,E2 9126.58} C_VEL
LIN {X 0,Y 283.555,Z 868.403,A -85,B 0,C 180,E1 9124.582,E2 9124.582} C_VEL
LIN {X 0,Y 273.109,Z 886.909,A -85,B 0,C 180,E1 9122.054,E2 9122.054} C_VEL
LIN {X 0,Y 263.175,Z 903.118,A -85,B 0,C 180,E1 9119.338,E2 9119.338} C_VEL
LIN {X 0,Y 252.623,Z 918.821,A -85,B 0,C 180,E1 9116.052,E2 9116.052} C_VEL
LIN {X 0,Y 242.373,Z 933.294,A -85,B 0,C 180,E1 9112.296,E2 9112.296} C_VEL
LIN {X 0,Y 233.061,Z 945.724,A -85,B 0,C 180,E1 9108.242,E2 9108.242} C_VEL
LIN {X 0,Y 223.608,Z 958.085,A -85,B 0,C 180,E1 9103.173,E2 9103.173} C_VEL
LIN {X 0,Y 216.362,Z 967.578,A -85,B 0,C 180,E1 9098.228,E2 9098.228} C_VEL
LIN {X 0,Y 209.956,Z 976.235,A -85,B 0,C 180,E1 9092.448,E2 9092.448} C_VEL
LIN {X 0,Y 205.614,Z 982.692,A -85,B 0,C 180,E1 9086.925,E2 9086.925} C_VEL
LIN {X 0,Y 202.416,Z 988.217,A -85,B 0,C 180,E1 9080.61,E2 9080.61} C_VEL
LIN {X 0,Y 200.848,Z 991.777,A -85,B 0,C 180,E1 9074.969,E2 9074.969} C_VEL
LIN {X 0,Y 200.175,Z 994.279,A -85,B 0,C 180,E1 9068.914,E2 9068.914} C_VEL
LIN {X 0,Y 200.03,Z 995.288,A -85,B 0,C 180,E1 9063.896,E2 9063.896} C_VEL
LIN {X 0,Y 200.06,Z 995.445,A -85,B 0,C 180,E1 9059.276,E2 9059.276} C_VEL
LIN {X 0,Y 200.254,Z 994.771,A -85,B 0,C 180,E1 9054.246,E2 9054.246} C_VEL
LIN {X 0,Y 201.188,Z 992.69,A -85,B 0,C 180,E1 9047.852,E2 9047.852} C_VEL
LIN {X 0,Y 203.312,Z 989.128,A -85,B 0,C 180,E1 9041.6,E2 9041.6} C_VEL
LIN {X 0,Y 207.376,Z 983.8,A -85,B 0,C 180,E1 9035.014,E2 9035.014} C_VEL
LIN {X 0,Y 212.923,Z 977.259,A -85,B 0,C 180,E1 9029.127,E2 9029.127} C_VEL
LIN {X 0,Y 221.332,Z 968,A -85,B 0,C 180,E1 9022.829,E2 9022.829} C_VEL
LIN {X 0,Y 230.757,Z 957.903,A -85,B 0,C 180,E1 9017.571,E2 9017.571} C_VEL
LIN {X 0,Y 241.21,Z 946.345,A -85,B 0,C 180,E1 9012.936,E2 9012.936} C_VEL
LIN {X 0,Y 252.927,Z 933.124,A -85,B 0,C 180,E1 9008.747,E2 9008.747} C_VEL
LIN {X 0,Y 264.147,Z 919.653,A -85,B 0,C 180,E1 9005.381,E2 9005.381} C_VEL
LIN {X 0,Y 277.591,Z 902.394,A -85,B 0,C 180,E1 9001.962,E2 9001.962} C_VEL
LIN {X 0,Y 290.271,Z 884.732,A -85,B 0,C 180,E1 8999.211,E2 8999.211} C_VEL
LIN {X 0,Y 302.026,Z 866.435,A -85,B 0,C 180,E1 8996.965,E2 8996.965} C_VEL
LIN {X 0,Y 307.516,Z 857.262,A -85,B 0,C 180,E1 8996.009,E2 8996.009} C_VEL
LIN {X 0,Y 310.7,Z 851.402,A -85,B 0,C 180,E1 8995.266,E2 8995.266} C_VEL
LIN {X 0,Y 317.224,Z 837.234,A -85,B 0,C 180,E1 8992.949,E2 8992.949} C_VEL
LIN {X 0,Y 320.173,Z 831.056,A -85,B 0,C 180,E1 8992.304,E2 8992.304} C_VEL
LIN {X 0,Y 330.06,Z 810.055,A -85,B 0,C 180,E1 8990.972,E2 8990.972} C_VEL
LIN {X 0,Y 338.163,Z 789.785,A -85,B 0,C 180,E1 8989.954,E2 8989.954} C_VEL
LIN {X 0,Y 345.863,Z 766.487,A -85,B 0,C 180,E1 8989.043,E2 8989.043} C_VEL
LIN {X 0,Y 351.141,Z 746.559,A -85,B 0,C 180,E1 8988.45,E2 8988.45} C_VEL
LIN {X 0,Y 355.92,Z 722.268,A -85,B 0,C 180,E1 8987.902,E2 8987.902} C_VEL
LIN {X 0,Y 368.594,Z 630.051,A -85,B 0,C 180,E1 8986.188,E2 8986.188} C_VEL
LIN {X 0,Y 355.022,Z 728.322,A -85,B 0,C 180,E1 8984.358,E2 8984.358} C_VEL
LIN {X 0,Y 349.985,Z 752.041,A -85,B 0,C 180,E1 8983.84,E2 8983.84} C_VEL
LIN {X 0,Y 343.381,Z 775.611,A -85,B 0,C 180,E1 8983.197,E2 8983.197} C_VEL
LIN {X 0,Y 336.553,Z 795.246,A -85,B 0,C 180,E1 8982.498,E2 8982.498} C_VEL
LIN {X 0,Y 327.499,Z 817.328,A -85,B 0,C 180,E1 8981.472,E2 8981.472} C_VEL
LIN {X 0,Y 317.675,Z 837.829,A -85,B 0,C 180,E1 8980.244,E2 8980.244} C_VEL
LIN {X 0,Y 306.052,Z 859.043,A -85,B 0,C 180,E1 8978.614,E2 8978.614} C_VEL
LIN {X 0,Y 294.376,Z 878.138,A -85,B 0,C 180,E1 8976.755,E2 8976.755} C_VEL
LIN {X 0,Y 281.938,Z 896.377,A -85,B 0,C 180,E1 8974.505,E2 8974.505} C_VEL
LIN {X 0,Y 268.975,Z 913.979,A -85,B 0,C 180,E1 8971.773,E2 8971.773} C_VEL
LIN {X 0,Y 256.383,Z 929.699,A -85,B 0,C 180,E1 8968.666,E2 8968.666} C_VEL
LIN {X 0,Y 242.798,Z 945.728,A -85,B 0,C 180,E1 8964.634,E2 8964.634} C_VEL
LIN {X 0,Y 230.586,Z 959.6,A -85,B 0,C 180,E1 8960.139,E2 8960.139} C_VEL
LIN {X 0,Y 219.4,Z 971.881,A -85,B 0,C 180,E1 8954.949,E2 8954.949} C_VEL
LIN {X 0,Y 209.703,Z 982.779,A -85,B 0,C 180,E1 8948.999,E2 8948.999} C_VEL
LIN {X 0,Y 202.757,Z 990.977,A -85,B 0,C 180,E1 8943.196,E2 8943.196} C_VEL
LIN {X 0,Y 197.046,Z 998.492,A -85,B 0,C 180,E1 8936.206,E2 8936.206} C_VEL
LIN {X 0,Y 193.977,Z 1003.546,A -85,B 0,C 180,E1 8929.898,E2 8929.898} C_VEL
LIN {X 0,Y 192.389,Z 1007.272,A -85,B 0,C 180,E1 8923.228,E2 8923.228} C_VEL
LIN {X 0,Y 192.01,Z 1009.174,A -85,B 0,C 180,E1 8917.79,E2 8917.79} C_VEL
LIN {X 0,Y 192.012,Z 1010.008,A -85,B 0,C 180,E1 8912.994,E2 8912.994} C_VEL
LIN {X 0,Y 192.041,Z 1010.008,A -85,B 0,C 180,E1 8908.219,E2 8908.219} C_VEL
LIN {X 0,Y 192.006,Z 1009.024,A -85,B 0,C 180,E1 8902.83,E2 8902.83} C_VEL
LIN {X 0,Y 192.436,Z 1006.425,A -85,B 0,C 180,E1 8896.488,E2 8896.488} C_VEL
LIN {X 0,Y 193.753,Z 1002.813,A -85,B 0,C 180,E1 8890.725,E2 8890.725} C_VEL
LIN {X 0,Y 196.968,Z 996.766,A -85,B 0,C 180,E1 8883.803,E2 8883.803} C_VEL
LIN {X 0,Y 201.468,Z 989.907,A -85,B 0,C 180,E1 8877.937,E2 8877.937} C_VEL
LIN {X 0,Y 208.32,Z 980.538,A -85,B 0,C 180,E1 8871.758,E2 8871.758} C_VEL
LIN {X 0,Y 216.245,Z 970.272,A -85,B 0,C 180,E1 8866.467,E2 8866.467} C_VEL
LIN {X 0,Y 225.71,Z 958.001,A -85,B 0,C 180,E1 8861.541,E2 8861.541} C_VEL
LIN {X 0,Y 236.012,Z 944.448,A -85,B 0,C 180,E1 8857.222,E2 8857.222} C_VEL
LIN {X 0,Y 246.199,Z 930.27,A -85,B 0,C 180,E1 8853.655,E2 8853.655} C_VEL
LIN {X 0,Y 257.439,Z 913.789,A -85,B 0,C 180,E1 8850.324,E2 8850.324} C_VEL
LIN {X 0,Y 267.616,Z 897.604,A -85,B 0,C 180,E1 8847.709,E2 8847.709} C_VEL
LIN {X 0,Y 278.884,Z 877.921,A -85,B 0,C 180,E1 8845.16,E2 8845.16} C_VEL
LIN {X 0,Y 288.74,Z 858.863,A -85,B 0,C 180,E1 8843.185,E2 8843.185} C_VEL
LIN {X 0,Y 297.726,Z 839.053,A -85,B 0,C 180,E1 8841.547,E2 8841.547} C_VEL
LIN {X 0,Y 306.112,Z 818.174,A -85,B 0,C 180,E1 8840.154,E2 8840.154} C_VEL
LIN {X 0,Y 313.105,Z 797.495,A -85,B 0,C 180,E1 8839.073,E2 8839.073} C_VEL
LIN {X 0,Y 319.666,Z 774.426,A -85,B 0,C 180,E1 8838.133,E2 8838.133} C_VEL
LIN {X 0,Y 324.571,Z 752.447,A -85,B 0,C 180,E1 8837.468,E2 8837.468} C_VEL
LIN {X 0,Y 328.478,Z 727.617,A -85,B 0,C 180,E1 8836.875,E2 8836.875} C_VEL
LIN {X 0,Y 344.126,Z 571.025,A -85,B 0,C 180,E1 8833.83,E2 8833.83} C_VEL
LIN {X 0,Y 338.308,Z 561.476,A -85,B 0,C 180,E1 8830.249,E2 8830.249} C_VEL
LIN {X 0,Y 334.148,Z 555.306,A -85,B 0,C 180,E1 8827.305,E2 8827.305} C_VEL
LIN {X 0,Y 331.739,Z 551.669,A -85,B 0,C 180,E1 8825.36,E2 8825.36} C_VEL
LIN {X 0,Y 328.946,Z 547.516,A -85,B 0,C 180,E1 8822.787,E2 8822.787} C_VEL
LIN {X 0,Y 325.856,Z 542.881,A -85,B 0,C 180,E1 8819.296,E2 8819.296} C_VEL
LIN {X 0,Y 323.107,Z 539.103,A -85,B 0,C 180,E1 8815.207,E2 8815.207} C_VEL
LIN {X 0,Y 322.557,Z 537.745,A -85,B 0,C 180,E1 8813.949,E2 8813.949} C_VEL
LIN {X 0,Y 320.504,Z 536.085,A -85,B 0,C 180,E1 8807.019,E2 8807.019} C_VEL
LIN {X 0,Y 320.729,Z 536.339,A -85,B 0,C 180,E1 8802.517,E2 8802.517} C_VEL
LIN {X 0,Y 322.757,Z 538.071,A -85,B 0,C 180,E1 8796.831,E2 8796.831} C_VEL
LIN {X 0,Y 325.372,Z 542.425,A -85,B 0,C 180,E1 8792.551,E2 8792.551} C_VEL
LIN {X 0,Y 326.405,Z 543.677,A -85,B 0,C 180,E1 8791.253,E2 8791.253} C_VEL
LIN {X 0,Y 329.999,Z 549.037,A -85,B 0,C 180,E1 8787.465,E2 8787.465} C_VEL
LIN {X 0,Y 333.43,Z 554.167,A -85,B 0,C 180,E1 8784.531,E2 8784.531} C_VEL
LIN {X 0,Y 337.17,Z 559.852,A -85,B 0,C 180,E1 8781.788,E2 8781.788} C_VEL
LIN {X 0,Y 342.761,Z 568.763,A -85,B 0,C 180,E1 8778.254,E2 8778.254} C_VEL
LIN {X 0,Y 343.71,Z 570.521,A -85,B 0,C 180,E1 8777.692,E2 8777.692} C_VEL
LIN {X 0,Y 328.627,Z 720.419,A -85,B 0,C 180,E1 8774.782,E2 8774.782} C_VEL
LIN {X 0,Y 324.686,Z 744.146,A -85,B 0,C 180,E1 8774.178,E2 8774.178} C_VEL
LIN {X 0,Y 319.873,Z 765.971,A -85,B 0,C 180,E1 8773.437,E2 8773.437} C_VEL
LIN {X 0,Y 313.804,Z 787.356,A -85,B 0,C 180,E1 8772.482,E2 8772.482} C_VEL
LIN {X 0,Y 306.719,Z 808.515,A -85,B 0,C 180,E1 8771.299,E2 8771.299} C_VEL
LIN {X 0,Y 298.625,Z 828.789,A -85,B 0,C 180,E1 8769.87,E2 8769.87} C_VEL
LIN {X 0,Y 288.939,Z 850.013,A -85,B 0,C 180,E1 8768.012,E2 8768.012} C_VEL
LIN {X 0,Y 279.53,Z 868.213,A -85,B 0,C 180,E1 8766.035,E2 8766.035} C_VEL
LIN {X 0,Y 268.773,Z 886.827,A -85,B 0,C 180,E1 8763.525,E2 8763.525} C_VEL
LIN {X 0,Y 258.193,Z 903.567,A -85,B 0,C 180,E1 8760.733,E2 8760.733} C_VEL
LIN {X 0,Y 247.274,Z 919.259,A -85,B 0,C 180,E1 8757.44,E2 8757.44} C_VEL
LIN {X 0,Y 236.626,Z 933.745,A -85,B 0,C 180,E1 8753.658,E2 8753.658} C_VEL
LIN {X 0,Y 226.924,Z 946.183,A -85,B 0,C 180,E1 8749.555,E2 8749.555} C_VEL
LIN {X 0,Y 217.019,Z 958.517,A -85,B 0,C 180,E1 8744.397,E2 8744.397} C_VEL
LIN {X 0,Y 209.402,Z 968.007,A -85,B 0,C 180,E1 8739.334,E2 8739.334} C_VEL
LIN {X 0,Y 202.627,Z 976.651,A -85,B 0,C 180,E1 8733.386,E2 8733.386} C_VEL
LIN {X 0,Y 197.81,Z 983.401,A -85,B 0,C 180,E1 8727.384,E2 8727.384} C_VEL
LIN {X 0,Y 194.466,Z 988.797,A -85,B 0,C 180,E1 8720.82,E2 8720.82} C_VEL
LIN {X 0,Y 192.797,Z 992.454,A -85,B 0,C 180,E1 8714.655,E2 8714.655} C_VEL
LIN {X 0,Y 192.144,Z 994.753,A -85,B 0,C 180,E1 8708.309,E2 8708.309} C_VEL
LIN {X 0,Y 192.036,Z 995.628,A -85,B 0,C 180,E1 8703.39,E2 8703.39} C_VEL
LIN {X 0,Y 192.088,Z 995.727,A -85,B 0,C 180,E1 8698.614,E2 8698.614} C_VEL
LIN {X 0,Y 192.346,Z 994.964,A -85,B 0,C 180,E1 8693.182,E2 8693.182} C_VEL
LIN {X 0,Y 193.492,Z 992.746,A -85,B 0,C 180,E1 8686.575,E2 8686.575} C_VEL
LIN {X 0,Y 195.855,Z 989.328,A -85,B 0,C 180,E1 8680.419,E2 8680.419} C_VEL
LIN {X 0,Y 200.408,Z 983.919,A -85,B 0,C 180,E1 8673.561,E2 8673.561} C_VEL
LIN {X 0,Y 206.881,Z 976.978,A -85,B 0,C 180,E1 8667.204,E2 8667.204} C_VEL
LIN {X 0,Y 215.507,Z 968.132,A -85,B 0,C 180,E1 8661.147,E2 8661.147} C_VEL
LIN {X 0,Y 225.549,Z 958.049,A -85,B 0,C 180,E1 8655.834,E2 8655.834} C_VEL
LIN {X 0,Y 236.987,Z 946.123,A -85,B 0,C 180,E1 8651.056,E2 8651.056} C_VEL
LIN {X 0,Y 250.073,Z 931.957,A -85,B 0,C 180,E1 8646.659,E2 8646.659} C_VEL
LIN {X 0,Y 263.113,Z 916.979,A -85,B 0,C 180,E1 8643.051,E2 8643.051} C_VEL
LIN {X 0,Y 276.077,Z 900.706,A -85,B 0,C 180,E1 8640.001,E2 8640.001} C_VEL
LIN {X 0,Y 289.291,Z 882.685,A -85,B 0,C 180,E1 8637.333,E2 8637.333} C_VEL
LIN {X 0,Y 300.028,Z 866.485,A -85,B 0,C 180,E1 8635.413,E2 8635.413} C_VEL
LIN {X 0,Y 311.977,Z 846.474,A -85,B 0,C 180,E1 8633.503,E2 8633.503} C_VEL
LIN {X 0,Y 320.173,Z 831.056,A -85,B 0,C 180,E1 8632.304,E2 8632.304} C_VEL
LIN {X 0,Y 323.229,Z 824.767,A -85,B 0,C 180,E1 8631.694,E2 8631.694} C_VEL
LIN {X 0,Y 329.618,Z 809.463,A -85,B 0,C 180,E1 8629.704,E2 8629.704} C_VEL
LIN {X 0,Y 332.332,Z 802.892,A -85,B 0,C 180,E1 8629.181,E2 8629.181} C_VEL
LIN {X 0,Y 340.877,Z 780.606,A -85,B 0,C 180,E1 8628.199,E2 8628.199} C_VEL
LIN {X 0,Y 347.637,Z 758.96,A -85,B 0,C 180,E1 8627.463,E2 8627.463} C_VEL
LIN {X 0,Y 353.154,Z 735.969,A -85,B 0,C 180,E1 8626.881,E2 8626.881} C_VEL
LIN {X 0,Y 357.304,Z 711.887,A -85,B 0,C 180,E1 8626.41,E2 8626.41} C_VEL
LIN {X 0,Y 358.947,Z 699.912,A -85,B 0,C 180,E1 8626.185,E2 8626.185} C_VEL
LIN {X 0,Y 353.848,Z 732.718,A -85,B 0,C 180,E1 8625.571,E2 8625.571} C_VEL
LIN {X 0,Y 348.694,Z 755.442,A -85,B 0,C 180,E1 8625.08,E2 8625.08} C_VEL
LIN {X 0,Y 341.726,Z 778.617,A -85,B 0,C 180,E1 8624.452,E2 8624.452} C_VEL
LIN {X 0,Y 334.362,Z 798.896,A -85,B 0,C 180,E1 8623.731,E2 8623.731} C_VEL
LIN {X 0,Y 325.103,Z 820.098,A -85,B 0,C 180,E1 8622.746,E2 8622.746} C_VEL
LIN {X 0,Y 314.548,Z 841.253,A -85,B 0,C 180,E1 8621.484,E2 8621.484} C_VEL
LIN {X 0,Y 302.764,Z 861.613,A -85,B 0,C 180,E1 8619.913,E2 8619.913} C_VEL
LIN {X 0,Y 289.318,Z 882.367,A -85,B 0,C 180,E1 8617.858,E2 8617.858} C_VEL
LIN {X 0,Y 277.11,Z 899.4,A -85,B 0,C 180,E1 8615.712,E2 8615.712} C_VEL
LIN {X 0,Y 263.752,Z 916.47,A -85,B 0,C 180,E1 8612.992,E2 8612.992} C_VEL
LIN {X 0,Y 250.557,Z 932.226,A -85,B 0,C 180,E1 8609.815,E2 8609.815} C_VEL
LIN {X 0,Y 237.478,Z 946.743,A -85,B 0,C 180,E1 8606.05,E2 8606.05} C_VEL
LIN {X 0,Y 224.777,Z 960.358,A -85,B 0,C 180,E1 8601.535,E2 8601.535} C_VEL
LIN {X 0,Y 213.523,Z 972.006,A -85,B 0,C 180,E1 8596.502,E2 8596.502} C_VEL
LIN {X 0,Y 202.837,Z 983.189,A -85,B 0,C 180,E1 8590.179,E2 8590.179} C_VEL
LIN {X 0,Y 194.917,Z 991.97,A -85,B 0,C 180,E1 8583.651,E2 8583.651} C_VEL
LIN {X 0,Y 189.227,Z 998.848,A -85,B 0,C 180,E1 8576.697,E2 8576.697} C_VEL
LIN {X 0,Y 185.88,Z 1004.011,A -85,B 0,C 180,E1 8569.727,E2 8569.727} C_VEL
LIN {X 0,Y 184.375,Z 1007.266,A -85,B 0,C 180,E1 8563.175,E2 8563.175} C_VEL
LIN {X 0,Y 184.005,Z 1009.054,A -85,B 0,C 180,E1 8557.503,E2 8557.503} C_VEL
LIN {X 0,Y 184.041,Z 1009.832,A -85,B 0,C 180,E1 8551.877,E2 8551.877} C_VEL
LIN {X 0,Y 184.019,Z 1009.513,A -85,B 0,C 180,E1 8546.271,E2 8546.271} C_VEL
LIN {X 0,Y 184.084,Z 1008.058,A -85,B 0,C 180,E1 8540.632,E2 8540.632} C_VEL
LIN {X 0,Y 184.674,Z 1005.547,A -85,B 0,C 180,E1 8534.947,E2 8534.947} C_VEL
LIN {X 0,Y 186.579,Z 1001.303,A -85,B 0,C 180,E1 8528.31,E2 8528.31} C_VEL
LIN {X 0,Y 190.169,Z 995.338,A -85,B 0,C 180,E1 8521.77,E2 8521.77} C_VEL
LIN {X 0,Y 195.737,Z 987.709,A -85,B 0,C 180,E1 8515.325,E2 8515.325} C_VEL
LIN {X 0,Y 202.943,Z 978.517,A -85,B 0,C 180,E1 8509.446,E2 8509.446} C_VEL
LIN {X 0,Y 212.565,Z 966.686,A -85,B 0,C 180,E1 8503.597,E2 8503.597} C_VEL
LIN {X 0,Y 222.368,Z 954.594,A -85,B 0,C 180,E1 8498.948,E2 8498.948} C_VEL
LIN {X 0,Y 233.166,Z 940.708,A -85,B 0,C 180,E1 8494.772,E2 8494.772} C_VEL
LIN {X 0,Y 244.263,Z 925.809,A -85,B 0,C 180,E1 8491.201,E2 8491.201} C_VEL
LIN {X 0,Y 255.505,Z 909.363,A -85,B 0,C 180,E1 8488.104,E2 8488.104} C_VEL
LIN {X 0,Y 266.947,Z 891.26,A -85,B 0,C 180,E1 8485.375,E2 8485.375} C_VEL
LIN {X 0,Y 276.959,Z 873.762,A -85,B 0,C 180,E1 8483.267,E2 8483.267} C_VEL
LIN {X 0,Y 287.516,Z 853.142,A -85,B 0,C 180,E1 8481.276,E2 8481.276} C_VEL
LIN {X 0,Y 296.661,Z 832.921,A -85,B 0,C 180,E1 8479.721,E2 8479.721} C_VEL
LIN {X 0,Y 305.034,Z 811.214,A -85,B 0,C 180,E1 8478.413,E2 8478.413} C_VEL
LIN {X 0,Y 312.387,Z 788.829,A -85,B 0,C 180,E1 8477.355,E2 8477.355} C_VEL
LIN {X 0,Y 318.125,Z 767.326,A -85,B 0,C 180,E1 8476.589,E2 8476.589} C_VEL
LIN {X 0,Y 323.222,Z 742.383,A -85,B 0,C 180,E1 8475.912,E2 8475.912} C_VEL
LIN {X 0,Y 326.479,Z 718.587,A -85,B 0,C 180,E1 8475.39,E2 8475.39} C_VEL
LIN {X 0,Y 340.926,Z 576.214,A -85,B 0,C 180,E1 8472.663,E2 8472.663} C_VEL
LIN {X 0,Y 335.514,Z 567.463,A -85,B 0,C 180,E1 8469.173,E2 8469.173} C_VEL
LIN {X 0,Y 330.933,Z 560.193,A -85,B 0,C 180,E1 8465.634,E2 8465.634} C_VEL
LIN {X 0,Y 327.488,Z 555.168,A -85,B 0,C 180,E1 8462.449,E2 8462.449} C_VEL
LIN {X 0,Y 324.447,Z 550.585,A -85,B 0,C 180,E1 8458.94,E2 8458.94} C_VEL
LIN {X 0,Y 321.823,Z 546.734,A -85,B 0,C 180,E1 8454.83,E2 8454.83} C_VEL
LIN {X 0,Y 321.354,Z 545.626,A -85,B 0,C 180,E1 8453.747,E2 8453.747} C_VEL
LIN {X 0,Y 319.414,Z 544.008,A -85,B 0,C 180,E1 8446.974,E2 8446.974} C_VEL
LIN {X 0,Y 319.641,Z 544.268,A -85,B 0,C 180,E1 8442.524,E2 8442.524} C_VEL
LIN {X 0,Y 321.595,Z 546.023,A -85,B 0,C 180,E1 8436.948,E2 8436.948} C_VEL
LIN {X 0,Y 324.198,Z 550.337,A -85,B 0,C 180,E1 8432.634,E2 8432.634} C_VEL
LIN {X 0,Y 325.21,Z 551.71,A -85,B 0,C 180,E1 8431.338,E2 8431.338} C_VEL
LIN {X 0,Y 328.531,Z 556.707,A -85,B 0,C 180,E1 8427.773,E2 8427.773} C_VEL
LIN {X 0,Y 331.848,Z 561.773,A -85,B 0,C 180,E1 8424.866,E2 8424.866} C_VEL
LIN {X 0,Y 335.632,Z 567.627,A -85,B 0,C 180,E1 8422.035,E2 8422.035} C_VEL
LIN {X 0,Y 340.53,Z 575.612,A -85,B 0,C 180,E1 8418.864,E2 8418.864} C_VEL
LIN {X 0,Y 325.533,Z 720.776,A -85,B 0,C 180,E1 8416.073,E2 8416.073} C_VEL
LIN {X 0,Y 321.489,Z 744.598,A -85,B 0,C 180,E1 8415.476,E2 8415.476} C_VEL
LIN {X 0,Y 316.432,Z 766.973,A -85,B 0,C 180,E1 8414.726,E2 8414.726} C_VEL
LIN {X 0,Y 310.271,Z 788.172,A -85,B 0,C 180,E1 8413.792,E2 8413.792} C_VEL
LIN {X 0,Y 302.813,Z 809.82,A -85,B 0,C 180,E1 8412.591,E2 8412.591} C_VEL
LIN {X 0,Y 294.918,Z 829.173,A -85,B 0,C 180,E1 8411.245,E2 8411.245} C_VEL
LIN {X 0,Y 284.99,Z 850.389,A -85,B 0,C 180,E1 8409.412,E2 8409.412} C_VEL
LIN {X 0,Y 275.33,Z 868.591,A -85,B 0,C 180,E1 8407.455,E2 8407.455} C_VEL
LIN {X 0,Y 264.269,Z 887.211,A -85,B 0,C 180,E1 8404.964,E2 8404.964} C_VEL
LIN {X 0,Y 253.365,Z 903.985,A -85,B 0,C 180,E1 8402.182,E2 8402.182} C_VEL
LIN {X 0,Y 242.076,Z 919.692,A -85,B 0,C 180,E1 8398.888,E2 8398.888} C_VEL
LIN {X 0,Y 230.457,Z 934.843,A -85,B 0,C 180,E1 8394.879,E2 8394.879} C_VEL
LIN {X 0,Y 220.404,Z 947.222,A -85,B 0,C 180,E1 8390.713,E2 8390.713} C_VEL
LIN {X 0,Y 210.532,Z 958.942,A -85,B 0,C 180,E1 8385.697,E2 8385.697} C_VEL
LIN {X 0,Y 202.241,Z 968.776,A -85,B 0,C 180,E1 8380.31,E2 8380.31} C_VEL
LIN {X 0,Y 195.354,Z 977.044,A -85,B 0,C 180,E1 8374.394,E2 8374.394} C_VEL
LIN {X 0,Y 190.018,Z 984.089,A -85,B 0,C 180,E1 8367.88,E2 8367.88} C_VEL
LIN {X 0,Y 186.638,Z 989.163,A -85,B 0,C 180,E1 8361.364,E2 8361.364} C_VEL
LIN {X 0,Y 184.847,Z 992.808,A -85,B 0,C 180,E1 8354.942,E2 8354.942} C_VEL
LIN {X 0,Y 184.167,Z 995.003,A -85,B 0,C 180,E1 8348.66,E2 8348.66} C_VEL
LIN {X 0,Y 184.041,Z 995.912,A -85,B 0,C 180,E1 8343.536,E2 8343.536} C_VEL
LIN {X 0,Y 184.094,Z 996.044,A -85,B 0,C 180,E1 8338.509,E2 8338.509} C_VEL
LIN {X 0,Y 184.381,Z 995.32,A -85,B 0,C 180,E1 8332.861,E2 8332.861} C_VEL
LIN {X 0,Y 185.649,Z 993.177,A -85,B 0,C 180,E1 8325.981,E2 8325.981} C_VEL
LIN {X 0,Y 188.224,Z 989.83,A -85,B 0,C 180,E1 8319.603,E2 8319.603} C_VEL
LIN {X 0,Y 193.181,Z 984.484,A -85,B 0,C 180,E1 8312.459,E2 8312.459} C_VEL
LIN {X 0,Y 199.85,Z 977.85,A -85,B 0,C 180,E1 8306.122,E2 8306.122} C_VEL
LIN {X 0,Y 209.277,Z 968.89,A -85,B 0,C 180,E1 8299.727,E2 8299.727} C_VEL
LIN {X 0,Y 220.17,Z 958.613,A -85,B 0,C 180,E1 8294.197,E2 8294.197} C_VEL
LIN {X 0,Y 232.167,Z 946.809,A -85,B 0,C 180,E1 8289.42,E2 8289.42} C_VEL
LIN {X 0,Y 245.467,Z 933.158,A -85,B 0,C 180,E1 8285.142,E2 8285.142} C_VEL
LIN {X 0,Y 258.53,Z 918.808,A -85,B 0,C 180,E1 8281.666,E2 8281.666} C_VEL
LIN {X 0,Y 272.061,Z 902.675,A -85,B 0,C 180,E1 8278.614,E2 8278.614} C_VEL
LIN {X 0,Y 285.158,Z 885.736,A -85,B 0,C 180,E1 8276.08,E2 8276.08} C_VEL
LIN {X 0,Y 297.232,Z 868.267,A -85,B 0,C 180,E1 8274.015,E2 8274.015} C_VEL
LIN {X 0,Y 309.573,Z 848.47,A -85,B 0,C 180,E1 8272.146,E2 8272.146} C_VEL
LIN {X 0,Y 320.191,Z 829.013,A -85,B 0,C 180,E1 8270.689,E2 8270.689} C_VEL
LIN {X 0,Y 330.17,Z 807.925,A -85,B 0,C 180,E1 8269.435,E2 8269.435} C_VEL
LIN {X 0,Y 332.332,Z 802.892,A -85,B 0,C 180,E1 8269.181,E2 8269.181} C_VEL
LIN {X 0,Y 335.07,Z 796.214,A -85,B 0,C 180,E1 8268.688,E2 8268.688} C_VEL
LIN {X 0,Y 340.932,Z 779.859,A -85,B 0,C 180,E1 8266.976,E2 8266.976} C_VEL
LIN {X 0,Y 343.323,Z 772.938,A -85,B 0,C 180,E1 8266.56,E2 8266.56} C_VEL
LIN {X 0,Y 346.339,Z 763.064,A -85,B 0,C 180,E1 8266.229,E2 8266.229} C_VEL
LIN {X 0,Y 339.111,Z 785.279,A -85,B 0,C 180,E1 8265.609,E2 8265.609} C_VEL
LIN {X 0,Y 330.521,Z 806.59,A -85,B 0,C 180,E1 8264.809,E2 8264.809} C_VEL
LIN {X 0,Y 320.724,Z 827.581,A -85,B 0,C 180,E1 8263.791,E2 8263.791} C_VEL
LIN {X 0,Y 310.189,Z 846.852,A -85,B 0,C 180,E1 8262.589,E2 8262.589} C_VEL
LIN {X 0,Y 298.171,Z 866.629,A -85,B 0,C 180,E1 8261.031,E2 8261.031} C_VEL
LIN {X 0,Y 285.197,Z 885.447,A -85,B 0,C 180,E1 8259.128,E2 8259.128} C_VEL
LIN {X 0,Y 270.272,Z 905.061,A -85,B 0,C 180,E1 8256.569,E2 8256.569} C_VEL
LIN {X 0,Y 256.407,Z 921.739,A -85,B 0,C 180,E1 8253.762,E2 8253.762} C_VEL
LIN {X 0,Y 241.857,Z 937.79,A -85,B 0,C 180,E1 8250.256,E2 8250.256} C_VEL
LIN {X 0,Y 227.76,Z 952.497,A -85,B 0,C 180,E1 8246.078,E2 8246.078} C_VEL
LIN {X 0,Y 215.036,Z 965.14,A -85,B 0,C 180,E1 8241.376,E2 8241.376} C_VEL
LIN {X 0,Y 202.881,Z 976.941,A -85,B 0,C 180,E1 8235.589,E2 8235.589} C_VEL
LIN {X 0,Y 193.339,Z 986.414,A -85,B 0,C 180,E1 8229.511,E2 8229.511} C_VEL
LIN {X 0,Y 185.591,Z 994.38,A -85,B 0,C 180,E1 8222.608,E2 8222.608} C_VEL
LIN {X 0,Y 180.278,Z 1000.721,A -85,B 0,C 180,E1 8215.291,E2 8215.291} C_VEL
LIN {X 0,Y 177.425,Z 1004.946,A -85,B 0,C 180,E1 8208.406,E2 8208.406} C_VEL
LIN {X 0,Y 176.188,Z 1007.893,A -85,B 0,C 180,E1 8201.466,E2 8201.466} C_VEL
LIN {X 0,Y 176.011,Z 1009.24,A -85,B 0,C 180,E1 8195.225,E2 8195.225} C_VEL
LIN {X 0,Y 176.061,Z 1009.498,A -85,B 0,C 180,E1 8190.01,E2 8190.01} C_VEL
LIN {X 0,Y 176.022,Z 1008.906,A -85,B 0,C 180,E1 8184.796,E2 8184.796} C_VEL
LIN {X 0,Y 176.128,Z 1007.459,A -85,B 0,C 180,E1 8179.544,E2 8179.544} C_VEL
LIN {X 0,Y 176.985,Z 1004.655,A -85,B 0,C 180,E1 8173.266,E2 8173.266} C_VEL
LIN {X 0,Y 179.577,Z 999.722,A -85,B 0,C 180,E1 8165.938,E2 8165.938} C_VEL
LIN {X 0,Y 183.87,Z 993.54,A -85,B 0,C 180,E1 8159.222,E2 8159.222} C_VEL
LIN {X 0,Y 190.452,Z 985.195,A -85,B 0,C 180,E1 8152.497,E2 8152.497} C_VEL
LIN {X 0,Y 198.865,Z 975.326,A -85,B 0,C 180,E1 8146.385,E2 8146.385} C_VEL
LIN {X 0,Y 208.503,Z 964.028,A -85,B 0,C 180,E1 8141.068,E2 8141.068} C_VEL
LIN {X 0,Y 220.083,Z 950.221,A -85,B 0,C 180,E1 8136.05,E2 8136.05} C_VEL
LIN {X 0,Y 231.298,Z 936.256,A -85,B 0,C 180,E1 8132.102,E2 8132.102} C_VEL
LIN {X 0,Y 242.752,Z 920.903,A -85,B 0,C 180,E1 8128.699,E2 8128.699} C_VEL
LIN {X 0,Y 254.242,Z 904.477,A -85,B 0,C 180,E1 8125.785,E2 8125.785} C_VEL
LIN {X 0,Y 265.542,Z 886.484,A -85,B 0,C 180,E1 8123.279,E2 8123.279} C_VEL
LIN {X 0,Y 276.918,Z 866.462,A -85,B 0,C 180,E1 8121.059,E2 8121.059} C_VEL
LIN {X 0,Y 286.724,Z 847.014,A -85,B 0,C 180,E1 8119.346,E2 8119.346} C_VEL
LIN {X 0,Y 295.906,Z 826.094,A -85,B 0,C 180,E1 8117.884,E2 8117.884} C_VEL
LIN {X 0,Y 304.212,Z 804.255,A -85,B 0,C 180,E1 8116.677,E2 8116.677} C_VEL
LIN {X 0,Y 311.08,Z 782.219,A -85,B 0,C 180,E1 8115.743,E2 8115.743} C_VEL
LIN {X 0,Y 317.241,Z 757.785,A -85,B 0,C 180,E1 8114.972,E2 8114.972} C_VEL
LIN {X 0,Y 321.46,Z 735.039,A -85,B 0,C 180,E1 8114.416,E2 8114.416} C_VEL
LIN {X 0,Y 325.604,Z 698.698,A -85,B 0,C 180,E1 8113.69,E2 8113.69} C_VEL
LIN {X 0,Y 337.774,Z 581.519,A -85,B 0,C 180,E1 8111.478,E2 8111.478} C_VEL
LIN {X 0,Y 332.786,Z 573.251,A -85,B 0,C 180,E1 8108.03,E2 8108.03} C_VEL
LIN {X 0,Y 328.716,Z 566.929,A -85,B 0,C 180,E1 8104.71,E2 8104.71} C_VEL
LIN {X 0,Y 326.032,Z 562.818,A -85,B 0,C 180,E1 8102.108,E2 8102.108} C_VEL
LIN {X 0,Y 323.19,Z 558.42,A -85,B 0,C 180,E1 8098.758,E2 8098.758} C_VEL
LIN {X 0,Y 320.622,Z 554.576,A -85,B 0,C 180,E1 8094.631,E2 8094.631} C_VEL
LIN {X 0,Y 320.149,Z 553.507,A -85,B 0,C 180,E1 8093.544,E2 8093.544} C_VEL
LIN {X 0,Y 318.311,Z 551.911,A -85,B 0,C 180,E1 8086.743,E2 8086.743} C_VEL
LIN {X 0,Y 318.626,Z 552.294,A -85,B 0,C 180,E1 8082.089,E2 8082.089} C_VEL
LIN {X 0,Y 320.406,Z 553.884,A -85,B 0,C 180,E1 8077.137,E2 8077.137} C_VEL
LIN {X 0,Y 323.101,Z 558.321,A -85,B 0,C 180,E1 8072.625,E2 8072.625} C_VEL
LIN {X 0,Y 324.088,Z 559.872,A -85,B 0,C 180,E1 8071.331,E2 8071.331} C_VEL
LIN {X 0,Y 327.084,Z 564.401,A -85,B 0,C 180,E1 8068.072,E2 8068.072} C_VEL
LIN {X 0,Y 330.278,Z 569.378,A -85,B 0,C 180,E1 8065.203,E2 8065.203} C_VEL
LIN {X 0,Y 334.256,Z 575.628,A -85,B 0,C 180,E1 8062.177,E2 8062.177} C_VEL
LIN {X 0,Y 337.405,Z 580.995,A -85,B 0,C 180,E1 8060.045,E2 8060.045} C_VEL
LIN {X 0,Y 322.606,Z 721.122,A -85,B 0,C 180,E1 8057.389,E2 8057.389} C_VEL
LIN {X 0,Y 318.508,Z 744.78,A -85,B 0,C 180,E1 8056.807,E2 8056.807} C_VEL
LIN {X 0,Y 313.349,Z 767.179,A -85,B 0,C 180,E1 8056.072,E2 8056.072} C_VEL
LIN {X 0,Y 307.005,Z 788.567,A -85,B 0,C 180,E1 8055.148,E2 8055.148} C_VEL
LIN {X 0,Y 299.443,Z 810.054,A -85,B 0,C 180,E1 8053.979,E2 8053.979} C_VEL
LIN {X 0,Y 290.992,Z 830.281,A -85,B 0,C 180,E1 8052.591,E2 8052.591} C_VEL
LIN {X 0,Y 280.838,Z 851.399,A -85,B 0,C 180,E1 8050.781,E2 8050.781} C_VEL
LIN {X 0,Y 270.946,Z 869.582,A -85,B 0,C 180,E1 8048.844,E2 8048.844} C_VEL
LIN {X 0,Y 259.937,Z 887.581,A -85,B 0,C 180,E1 8046.452,E2 8046.452} C_VEL
LIN {X 0,Y 248.699,Z 904.354,A -85,B 0,C 180,E1 8043.688,E2 8043.688} C_VEL
LIN {X 0,Y 237.031,Z 920.063,A -85,B 0,C 180,E1 8040.401,E2 8040.401} C_VEL
LIN {X 0,Y 225.554,Z 934.555,A -85,B 0,C 180,E1 8036.588,E2 8036.588} C_VEL
LIN {X 0,Y 215.02,Z 947.015,A -85,B 0,C 180,E1 8032.405,E2 8032.405} C_VEL
LIN {X 0,Y 204.159,Z 959.334,A -85,B 0,C 180,E1 8027.079,E2 8027.079} C_VEL
LIN {X 0,Y 195.345,Z 969.276,A -85,B 0,C 180,E1 8021.505,E2 8021.505} C_VEL
LIN {X 0,Y 187.836,Z 977.783,A -85,B 0,C 180,E1 8015.182,E2 8015.182} C_VEL
LIN {X 0,Y 182.238,Z 984.724,A -85,B 0,C 180,E1 8008.419,E2 8008.419} C_VEL
LIN {X 0,Y 178.699,Z 989.73,A -85,B 0,C 180,E1 8001.626,E2 8001.626} C_VEL
LIN {X 0,Y 176.786,Z 993.448,A -85,B 0,C 180,E1 7994.575,E2 7994.575} C_VEL
LIN {X 0,Y 176.156,Z 995.398,A -85,B 0,C 180,E1 7988.34,E2 7988.34} C_VEL
LIN {X 0,Y 176.048,Z 996.253,A -85,B 0,C 180,E1 7982.966,E2 7982.966} C_VEL
LIN {X 0,Y 176.108,Z 996.331,A -85,B 0,C 180,E1 7977.735,E2 7977.735} C_VEL
LIN {X 0,Y 176.551,Z 995.482,A -85,B 0,C 180,E1 7971.403,E2 7971.403} C_VEL
LIN {X 0,Y 178.254,Z 993.055,A -85,B 0,C 180,E1 7964.072,E2 7964.072} C_VEL
LIN {X 0,Y 181.74,Z 989.231,A -85,B 0,C 180,E1 7956.848,E2 7956.848} C_VEL
LIN {X 0,Y 187.549,Z 983.568,A -85,B 0,C 180,E1 7949.644,E2 7949.644} C_VEL
LIN {X 0,Y 195.547,Z 976.477,A -85,B 0,C 180,E1 7943.003,E2 7943.003} C_VEL
LIN {X 0,Y 205.485,Z 967.631,A -85,B 0,C 180,E1 7936.976,E2 7936.976} C_VEL
LIN {X 0,Y 218.137,Z 956.294,A -85,B 0,C 180,E1 7931.187,E2 7931.187} C_VEL
LIN {X 0,Y 231.447,Z 943.918,A -85,B 0,C 180,E1 7926.435,E2 7926.435} C_VEL
LIN {X 0,Y 245.641,Z 929.681,A -85,B 0,C 180,E1 7922.334,E2 7922.334} C_VEL
LIN {X 0,Y 260.533,Z 913.609,A -85,B 0,C 180,E1 7918.791,E2 7918.791} C_VEL
LIN {X 0,Y 274.284,Z 897.486,A -85,B 0,C 180,E1 7916.029,E2 7916.029} C_VEL
LIN {X 0,Y 287.727,Z 879.883,A -85,B 0,C 180,E1 7913.68,E2 7913.68} C_VEL
LIN {X 0,Y 300.229,Z 861.865,A -85,B 0,C 180,E1 7911.768,E2 7911.768} C_VEL
LIN {X 0,Y 311.573,Z 843.378,A -85,B 0,C 180,E1 7910.208,E2 7910.208} C_VEL
LIN {X 0,Y 323.211,Z 821.742,A -85,B 0,C 180,E1 7908.762,E2 7908.762} C_VEL
LIN {X 0,Y 331.496,Z 803.895,A -85,B 0,C 180,E1 7907.812,E2 7907.812} C_VEL
LIN {X 0,Y 340.385,Z 781.407,A -85,B 0,C 180,E1 7906.858,E2 7906.858} C_VEL
LIN {X 0,Y 343.323,Z 772.938,A -85,B 0,C 180,E1 7906.56,E2 7906.56} C_VEL
LIN {X 0,Y 342.733,Z 774.725,A -85,B 0,C 180,E1 7906.407,E2 7906.407} C_VEL
LIN {X 0,Y 339.304,Z 784.492,A -85,B 0,C 180,E1 7906.296,E2 7906.296} C_VEL
LIN {X 0,Y 332.286,Z 802.206,A -85,B 0,C 180,E1 7906.47,E2 7906.47} C_VEL
LIN {X 0,Y 327.351,Z 812.965,A -85,B 0,C 180,E1 7906.819,E2 7906.819} C_VEL
LIN {X 0,Y 326.917,Z 813.833,A -85,B 0,C 180,E1 7906.862,E2 7906.862} C_VEL
LIN {X 0,Y 316.082,Z 834.593,A -85,B 0,C 180,E1 7908.065,E2 7908.065} C_VEL
LIN {X 0,Y 303.5,Z 855.54,A -85,B 0,C 180,E1 7909.612,E2 7909.612} C_VEL
LIN {X 0,Y 291.685,Z 872.932,A -85,B 0,C 180,E1 7911.237,E2 7911.237} C_VEL
LIN {X 0,Y 277.767,Z 891.162,A -85,B 0,C 180,E1 7913.386,E2 7913.386} C_VEL
LIN {X 0,Y 263.307,Z 908.315,A -85,B 0,C 180,E1 7915.972,E2 7915.972} C_VEL
LIN {X 0,Y 248.468,Z 924.122,A -85,B 0,C 180,E1 7919.079,E2 7919.079} C_VEL
LIN {X 0,Y 233.126,Z 939.165,A -85,B 0,C 180,E1 7922.951,E2 7922.951} C_VEL
LIN {X 0,Y 219.678,Z 951.495,A -85,B 0,C 180,E1 7927.105,E2 7927.105} C_VEL
LIN {X 0,Y 206.6,Z 962.675,A -85,B 0,C 180,E1 7932.121,E2 7932.121} C_VEL
LIN {X 0,Y 194.892,Z 972.435,A -85,B 0,C 180,E1 7937.929,E2 7937.929} C_VEL
LIN {X 0,Y 185.344,Z 980.241,A -85,B 0,C 180,E1 7944.243,E2 7944.243} C_VEL
LIN {X 0,Y 177.42,Z 986.917,A -85,B 0,C 180,E1 7951.668,E2 7951.668} C_VEL
LIN {X 0,Y 172.402,Z 991.556,A -85,B 0,C 180,E1 7958.987,E2 7958.987} C_VEL
LIN {X 0,Y 169.428,Z 994.734,A -85,B 0,C 180,E1 7966.787,E2 7966.787} C_VEL
LIN {X 0,Y 168.358,Z 996.236,A -85,B 0,C 180,E1 7973.3,E2 7973.3} C_VEL
LIN {X 0,Y 168.068,Z 996.765,A -85,B 0,C 180,E1 7980.007,E2 7980.007} C_VEL
LIN {X 0,Y 168.094,Z 996.133,A -85,B 0,C 180,E1 7986.355,E2 7986.355} C_VEL
LIN {X 0,Y 168.466,Z 994.618,A -85,B 0,C 180,E1 7992.371,E2 7992.371} C_VEL
LIN {X 0,Y 169.705,Z 992,A -85,B 0,C 180,E1 7998.779,E2 7998.779} C_VEL
LIN {X 0,Y 173.042,Z 987.122,A -85,B 0,C 180,E1 8006.678,E2 8006.678} C_VEL
LIN {X 0,Y 177.702,Z 981.499,A -85,B 0,C 180,E1 8013.216,E2 8013.216} C_VEL
LIN {X 0,Y 185.122,Z 973.312,A -85,B 0,C 180,E1 8020.257,E2 8020.257} C_VEL
LIN {X 0,Y 193.742,Z 964.234,A -85,B 0,C 180,E1 8026.172,E2 8026.172} C_VEL
LIN {X 0,Y 203.913,Z 953.242,A -85,B 0,C 180,E1 8031.567,E2 8031.567} C_VEL
LIN {X 0,Y 214.943,Z 941.08,A -85,B 0,C 180,E1 8036.216,E2 8036.216} C_VEL
LIN {X 0,Y 226.407,Z 927.541,A -85,B 0,C 180,E1 8040.218,E2 8040.218} C_VEL
LIN {X 0,Y 238.751,Z 911.934,A -85,B 0,C 180,E1 8043.837,E2 8043.837} C_VEL
LIN {X 0,Y 249.736,Z 896.81,A -85,B 0,C 180,E1 8046.612,E2 8046.612} C_VEL
LIN {X 0,Y 261.559,Z 878.873,A -85,B 0,C 180,E1 8049.236,E2 8049.236} C_VEL
LIN {X 0,Y 272.547,Z 860.398,A -85,B 0,C 180,E1 8051.4,E2 8051.4} C_VEL
LIN {X 0,Y 282.395,Z 841.507,A -85,B 0,C 180,E1 8053.165,E2 8053.165} C_VEL
LIN {X 0,Y 291.924,Z 820.864,A -85,B 0,C 180,E1 8054.726,E2 8054.726} C_VEL
LIN {X 0,Y 300.195,Z 799.631,A -85,B 0,C 180,E1 8055.997,E2 8055.997} C_VEL
LIN {X 0,Y 307.786,Z 776.373,A -85,B 0,C 180,E1 8057.09,E2 8057.09} C_VEL
LIN {X 0,Y 313.782,Z 753.63,A -85,B 0,C 180,E1 8057.913,E2 8057.913} C_VEL
LIN {X 0,Y 318.393,Z 730.137,A -85,B 0,C 180,E1 8058.533,E2 8058.533} C_VEL
LIN {X 0,Y 321.934,Z 703.378,A -85,B 0,C 180,E1 8059.078,E2 8059.078} C_VEL
LIN {X 0,Y 334.375,Z 586.269,A -85,B 0,C 180,E1 8061.271,E2 8061.271} C_VEL
LIN {X 0,Y 330.084,Z 579.097,A -85,B 0,C 180,E1 8064.437,E2 8064.437} C_VEL
LIN {X 0,Y 326.845,Z 574.031,A -85,B 0,C 180,E1 8067.216,E2 8067.216} C_VEL
LIN {X 0,Y 324.468,Z 570.26,A -85,B 0,C 180,E1 8069.621,E2 8069.621} C_VEL
LIN {X 0,Y 321.984,Z 566.283,A -85,B 0,C 180,E1 8072.639,E2 8072.639} C_VEL
LIN {X 0,Y 319.251,Z 561.843,A -85,B 0,C 180,E1 8077.244,E2 8077.244} C_VEL
LIN {X 0,Y 318.058,Z 560.742,A -85,B 0,C 180,E1 8080.152,E2 8080.152} C_VEL
LIN {X 0,Y 317.194,Z 559.762,A -85,B 0,C 180,E1 8085.393,E2 8085.393} C_VEL
LIN {X 0,Y 317.889,Z 560.608,A -85,B 0,C 180,E1 8090.586,E2 8090.586} C_VEL
LIN {X 0,Y 319.204,Z 561.767,A -85,B 0,C 180,E1 8093.886,E2 8093.886} C_VEL
LIN {X 0,Y 321.529,Z 565.84,A -85,B 0,C 180,E1 8098.039,E2 8098.039} C_VEL
LIN {X 0,Y 322.552,Z 567.261,A -85,B 0,C 180,E1 8099.378,E2 8099.378} C_VEL
LIN {X 0,Y 325.743,Z 572.275,A -85,B 0,C 180,E1 8102.99,E2 8102.99} C_VEL
LIN {X 0,Y 328.752,Z 577.06,A -85,B 0,C 180,E1 8105.759,E2 8105.759} C_VEL
LIN {X 0,Y 332.901,Z 583.681,A -85,B 0,C 180,E1 8108.985,E2 8108.985} C_VEL
LIN {X 0,Y 334.759,Z 587.069,A -85,B 0,C 180,E1 8110.284,E2 8110.284} C_VEL
LIN {X 0,Y 319.285,Z 730.383,A -85,B 0,C 180,E1 8112.976,E2 8112.976} C_VEL
LIN {X 0,Y 315.065,Z 754.191,A -85,B 0,C 180,E1 8113.53,E2 8113.53} C_VEL
LIN {X 0,Y 309.604,Z 776.869,A -85,B 0,C 180,E1 8114.184,E2 8114.184} C_VEL
LIN {X 0,Y 302.799,Z 798.923,A -85,B 0,C 180,E1 8115.048,E2 8115.048} C_VEL
LIN {X 0,Y 294.579,Z 821.229,A -85,B 0,C 180,E1 8116.175,E2 8116.175} C_VEL
LIN {X 0,Y 286.072,Z 840.887,A -85,B 0,C 180,E1 8117.441,E2 8117.441} C_VEL
LIN {X 0,Y 275.636,Z 861.856,A -85,B 0,C 180,E1 8119.144,E2 8119.144} C_VEL
LIN {X 0,Y 265.124,Z 880.571,A -85,B 0,C 180,E1 8121.054,E2 8121.054} C_VEL
LIN {X 0,Y 253.752,Z 898.559,A -85,B 0,C 180,E1 8123.374,E2 8123.374} C_VEL
LIN {X 0,Y 242.1,Z 915.46,A -85,B 0,C 180,E1 8126.09,E2 8126.09} C_VEL
LIN {X 0,Y 230.328,Z 930.93,A -85,B 0,C 180,E1 8129.264,E2 8129.264} C_VEL
LIN {X 0,Y 218.361,Z 945.692,A -85,B 0,C 180,E1 8133.095,E2 8133.095} C_VEL
LIN {X 0,Y 207.417,Z 958.361,A -85,B 0,C 180,E1 8137.325,E2 8137.325} C_VEL
LIN {X 0,Y 196.11,Z 970.993,A -85,B 0,C 180,E1 8142.778,E2 8142.778} C_VEL
LIN {X 0,Y 187.017,Z 981.131,A -85,B 0,C 180,E1 8148.489,E2 8148.489} C_VEL
LIN {X 0,Y 179.26,Z 989.935,A -85,B 0,C 180,E1 8155.075,E2 8155.075} C_VEL
LIN {X 0,Y 173.538,Z 997.188,A -85,B 0,C 180,E1 8162.193,E2 8162.193} C_VEL
LIN {X 0,Y 170.073,Z 1002.422,A -85,B 0,C 180,E1 8169.357,E2 8169.357} C_VEL
LIN {X 0,Y 168.394,Z 1006.256,A -85,B 0,C 180,E1 8176.622,E2 8176.622} C_VEL
LIN {X 0,Y 168.025,Z 1008.295,A -85,B 0,C 180,E1 8183.176,E2 8183.176} C_VEL
LIN {X 0,Y 168.059,Z 1009.11,A -85,B 0,C 180,E1 8188.647,E2 8188.647} C_VEL
LIN {X 0,Y 168.022,Z 1009.102,A -85,B 0,C 180,E1 8193.763,E2 8193.763} C_VEL
LIN {X 0,Y 168.073,Z 1008.279,A -85,B 0,C 180,E1 8199.253,E2 8199.253} C_VEL
LIN {X 0,Y 168.783,Z 1006.264,A -85,B 0,C 180,E1 8205.823,E2 8205.823} C_VEL
LIN {X 0,Y 171.381,Z 1002.294,A -85,B 0,C 180,E1 8213.748,E2 8213.748} C_VEL
LIN {X 0,Y 176.055,Z 996.935,A -85,B 0,C 180,E1 8221.129,E2 8221.129} C_VEL
LIN {X 0,Y 183.786,Z 989.281,A -85,B 0,C 180,E1 8228.739,E2 8228.739} C_VEL
LIN {X 0,Y 193.619,Z 980.287,A -85,B 0,C 180,E1 8235.389,E2 8235.389} C_VEL
LIN {X 0,Y 205.269,Z 969.6,A -85,B 0,C 180,E1 8241.212,E2 8241.212} C_VEL
LIN {X 0,Y 218.665,Z 957.225,A -85,B 0,C 180,E1 8246.337,E2 8246.337} C_VEL
LIN {X 0,Y 231.481,Z 944.808,A -85,B 0,C 180,E1 8250.261,E2 8250.261} C_VEL
LIN {X 0,Y 246.798,Z 929.086,A -85,B 0,C 180,E1 8254.09,E2 8254.09} C_VEL
LIN {X 0,Y 260.839,Z 913.604,A -85,B 0,C 180,E1 8256.985,E2 8256.985} C_VEL
LIN {X 0,Y 275.379,Z 896.053,A -85,B 0,C 180,E1 8259.526,E2 8259.526} C_VEL
LIN {X 0,Y 289.705,Z 877.115,A -85,B 0,C 180,E1 8261.654,E2 8261.654} C_VEL
LIN {X 0,Y 302.691,Z 857.728,A -85,B 0,C 180,E1 8263.335,E2 8263.335} C_VEL
LIN {X 0,Y 315.532,Z 836.083,A -85,B 0,C 180,E1 8264.787,E2 8264.787} C_VEL
LIN {X 0,Y 325.439,Z 816.94,A -85,B 0,C 180,E1 8265.783,E2 8265.783} C_VEL
LIN {X 0,Y 331.696,Z 803.301,A -85,B 0,C 180,E1 8266.362,E2 8266.362} C_VEL
LIN {X 0,Y 326.917,Z 813.833,A -85,B 0,C 180,E1 8266.862,E2 8266.862} C_VEL
LIN {X 0,Y 323.912,Z 819.819,A -85,B 0,C 180,E1 8267.011,E2 8267.011} C_VEL
LIN {X 0,Y 319.826,Z 827.771,A -85,B 0,C 180,E1 8266.841,E2 8266.841} C_VEL
LIN {X 0,Y 311.148,Z 843.068,A -85,B 0,C 180,E1 8265.89,E2 8265.89} C_VEL
LIN {X 0,Y 310.015,Z 844.928,A -85,B 0,C 180,E1 8265.768,E2 8265.768} C_VEL
LIN {X 0,Y 297.722,Z 864.211,A -85,B 0,C 180,E1 8264.416,E2 8264.416} C_VEL
LIN {X 0,Y 283.852,Z 883.36,A -85,B 0,C 180,E1 8262.68,E2 8262.68} C_VEL
LIN {X 0,Y 268.917,Z 901.991,A -85,B 0,C 180,E1 8260.495,E2 8260.495} C_VEL
LIN {X 0,Y 253.678,Z 919.096,A -85,B 0,C 180,E1 8257.869,E2 8257.869} C_VEL
LIN {X 0,Y 237.971,Z 935.264,A -85,B 0,C 180,E1 8254.613,E2 8254.613} C_VEL
LIN {X 0,Y 222.499,Z 950.115,A -85,B 0,C 180,E1 8250.679,E2 8250.679} C_VEL
LIN {X 0,Y 208.171,Z 962.87,A -85,B 0,C 180,E1 8246.142,E2 8246.142} C_VEL
LIN {X 0,Y 193.808,Z 975.236,A -85,B 0,C 180,E1 8240.248,E2 8240.248} C_VEL
LIN {X 0,Y 182.584,Z 984.795,A -85,B 0,C 180,E1 8234.076,E2 8234.076} C_VEL
LIN {X 0,Y 173.168,Z 992.936,A -85,B 0,C 180,E1 8226.916,E2 8226.916} C_VEL
LIN {X 0,Y 166.346,Z 999.468,A -85,B 0,C 180,E1 8219.146,E2 8219.146} C_VEL
LIN {X 0,Y 162.281,Z 1003.998,A -85,B 0,C 180,E1 8211.327,E2 8211.327} C_VEL
LIN {X 0,Y 160.476,Z 1006.908,A -85,B 0,C 180,E1 8204.074,E2 8204.074} C_VEL
LIN {X 0,Y 160.018,Z 1008.584,A -85,B 0,C 180,E1 8196.551,E2 8196.551} C_VEL
LIN {X 0,Y 160.059,Z 1008.903,A -85,B 0,C 180,E1 8190.727,E2 8190.727} C_VEL
LIN {X 0,Y 160.032,Z 1008.361,A -85,B 0,C 180,E1 8184.993,E2 8184.993} C_VEL
LIN {X 0,Y 160.15,Z 1006.957,A -85,B 0,C 180,E1 8179.216,E2 8179.216} C_VEL
LIN {X 0,Y 161.074,Z 1004.356,A -85,B 0,C 180,E1 8172.677,E2 8172.677} C_VEL
LIN {X 0,Y 163.955,Z 999.658,A -85,B 0,C 180,E1 8164.743,E2 8164.743} C_VEL
LIN {X 0,Y 168.529,Z 993.841,A -85,B 0,C 180,E1 8157.741,E2 8157.741} C_VEL
LIN {X 0,Y 176.218,Z 985.288,A -85,B 0,C 180,E1 8150.136,E2 8150.136} C_VEL
LIN {X 0,Y 184.937,Z 976.132,A -85,B 0,C 180,E1 8144.039,E2 8144.039} C_VEL
LIN {X 0,Y 195.38,Z 965.095,A -85,B 0,C 180,E1 8138.483,E2 8138.483} C_VEL
LIN {X 0,Y 206.733,Z 952.868,A -85,B 0,C 180,E1 8133.727,E2 8133.727} C_VEL
LIN {X 0,Y 219.032,Z 938.697,A -85,B 0,C 180,E1 8129.537,E2 8129.537} C_VEL
LIN {X 0,Y 231.806,Z 923.012,A -85,B 0,C 180,E1 8125.924,E2 8125.924} C_VEL
LIN {X 0,Y 243.477,Z 907.396,A -85,B 0,C 180,E1 8123.116,E2 8123.116} C_VEL
LIN {X 0,Y 256.111,Z 888.747,A -85,B 0,C 180,E1 8120.478,E2 8120.478} C_VEL
LIN {X 0,Y 267.579,Z 869.957,A -85,B 0,C 180,E1 8118.384,E2 8118.384} C_VEL
LIN {X 0,Y 278.096,Z 850.283,A -85,B 0,C 180,E1 8116.661,E2 8116.661} C_VEL
LIN {X 0,Y 287.993,Z 829.324,A -85,B 0,C 180,E1 8115.199,E2 8115.199} C_VEL
LIN {X 0,Y 296.457,Z 808.277,A -85,B 0,C 180,E1 8114.053,E2 8114.053} C_VEL
LIN {X 0,Y 304.3,Z 784.982,A -85,B 0,C 180,E1 8113.072,E2 8113.072} C_VEL
LIN {X 0,Y 310.609,Z 761.979,A -85,B 0,C 180,E1 8112.349,E2 8112.349} C_VEL
LIN {X 0,Y 315.316,Z 738.493,A -85,B 0,C 180,E1 8111.79,E2 8111.79} C_VEL
LIN {X 0,Y 319.095,Z 709.64,A -85,B 0,C 180,E1 8111.211,E2 8111.211} C_VEL
LIN {X 0,Y 331.805,Z 592.353,A -85,B 0,C 180,E1 8109.058,E2 8109.058} C_VEL
LIN {X 0,Y 328.022,Z 586.015,A -85,B 0,C 180,E1 8106.124,E2 8106.124} C_VEL
LIN {X 0,Y 325.312,Z 581.64,A -85,B 0,C 180,E1 8103.7,E2 8103.7} C_VEL
LIN {X 0,Y 323.106,Z 578.105,A -85,B 0,C 180,E1 8101.418,E2 8101.418} C_VEL
LIN {X 0,Y 320.55,Z 573.955,A -85,B 0,C 180,E1 8098.212,E2 8098.212} C_VEL
LIN {X 0,Y 318.116,Z 569.939,A -85,B 0,C 180,E1 8093.955,E2 8093.955} C_VEL
LIN {X 0,Y 317.666,Z 569.221,A -85,B 0,C 180,E1 8092.948,E2 8092.948} C_VEL
LIN {X 0,Y 316.119,Z 567.737,A -85,B 0,C 180,E1 8086.463,E2 8086.463} C_VEL
LIN {X 0,Y 316.549,Z 568.294,A -85,B 0,C 180,E1 8081.586,E2 8081.586} C_VEL
LIN {X 0,Y 318.062,Z 569.687,A -85,B 0,C 180,E1 8077.447,E2 8077.447} C_VEL
LIN {X 0,Y 320.805,Z 574.187,A -85,B 0,C 180,E1 8072.731,E2 8072.731} C_VEL
LIN {X 0,Y 324.233,Z 579.817,A -85,B 0,C 180,E1 8068.658,E2 8068.658} C_VEL
LIN {X 0,Y 327.273,Z 584.772,A -85,B 0,C 180,E1 8065.795,E2 8065.795} C_VEL
LIN {X 0,Y 331.183,Z 591.19,A -85,B 0,C 180,E1 8062.693,E2 8062.693} C_VEL
LIN {X 0,Y 331.455,Z 591.99,A -85,B 0,C 180,E1 8062.468,E2 8062.468} C_VEL
LIN {X 0,Y 317.14,Z 721.579,A -85,B 0,C 180,E1 8060.083,E2 8060.083} C_VEL
LIN {X 0,Y 312.866,Z 745.386,A -85,B 0,C 180,E1 8059.524,E2 8059.524} C_VEL
LIN {X 0,Y 307.485,Z 767.886,A -85,B 0,C 180,E1 8058.82,E2 8058.82} C_VEL
LIN {X 0,Y 300.925,Z 789.215,A -85,B 0,C 180,E1 8057.943,E2 8057.943} C_VEL
LIN {X 0,Y 292.764,Z 811.429,A -85,B 0,C 180,E1 8056.782,E2 8056.782} C_VEL
LIN {X 0,Y 284.024,Z 831.488,A -85,B 0,C 180,E1 8055.458,E2 8055.458} C_VEL
LIN {X 0,Y 273.408,Z 852.548,A -85,B 0,C 180,E1 8053.712,E2 8053.712} C_VEL
LIN {X 0,Y 262.658,Z 871.382,A -85,B 0,C 180,E1 8051.761,E2 8051.761} C_VEL
LIN {X 0,Y 251.247,Z 888.974,A -85,B 0,C 180,E1 8049.461,E2 8049.461} C_VEL
LIN {X 0,Y 239.186,Z 905.89,A -85,B 0,C 180,E1 8046.7,E2 8046.7} C_VEL
LIN {X 0,Y 227.463,Z 920.725,A -85,B 0,C 180,E1 8043.621,E2 8043.621} C_VEL
LIN {X 0,Y 215.121,Z 935.245,A -85,B 0,C 180,E1 8039.812,E2 8039.812} C_VEL
LIN {X 0,Y 203.694,Z 947.74,A -85,B 0,C 180,E1 8035.581,E2 8035.581} C_VEL
LIN {X 0,Y 191.801,Z 960.065,A -85,B 0,C 180,E1 8030.114,E2 8030.114} C_VEL
LIN {X 0,Y 182.022,Z 970.018,A -85,B 0,C 180,E1 8024.301,E2 8024.301} C_VEL
LIN {X 0,Y 173.582,Z 978.507,A -85,B 0,C 180,E1 8017.603,E2 8017.603} C_VEL
LIN {X 0,Y 167.21,Z 985.424,A -85,B 0,C 180,E1 8010.332,E2 8010.332} C_VEL
LIN {X 0,Y 163.169,Z 990.342,A -85,B 0,C 180,E1 8003.082,E2 8003.082} C_VEL
LIN {X 0,Y 160.953,Z 993.979,A -85,B 0,C 180,E1 7995.602,E2 7995.602} C_VEL
LIN {X 0,Y 160.172,Z 996.018,A -85,B 0,C 180,E1 7988.457,E2 7988.457} C_VEL
LIN {X 0,Y 160.058,Z 996.844,A -85,B 0,C 180,E1 7982.858,E2 7982.858} C_VEL
LIN {X 0,Y 160.135,Z 996.959,A -85,B 0,C 180,E1 7977.086,E2 7977.086} C_VEL
LIN {X 0,Y 160.685,Z 996.212,A -85,B 0,C 180,E1 7970.499,E2 7970.499} C_VEL
LIN {X 0,Y 162.759,Z 993.976,A -85,B 0,C 180,E1 7962.495,E2 7962.495} C_VEL
LIN {X 0,Y 166.53,Z 990.578,A -85,B 0,C 180,E1 7955.199,E2 7955.199} C_VEL
LIN {X 0,Y 173.761,Z 984.805,A -85,B 0,C 180,E1 7946.869,E2 7946.869} C_VEL
LIN {X 0,Y 183.017,Z 977.795,A -85,B 0,C 180,E1 7939.8,E2 7939.8} C_VEL
LIN {X 0,Y 194.362,Z 969.049,A -85,B 0,C 180,E1 7933.495,E2 7933.495} C_VEL
LIN {X 0,Y 207.344,Z 958.872,A -85,B 0,C 180,E1 7928.04,E2 7928.04} C_VEL
LIN {X 0,Y 221.022,Z 947.413,A -85,B 0,C 180,E1 7923.489,E2 7923.489} C_VEL
LIN {X 0,Y 237.009,Z 933.101,A -85,B 0,C 180,E1 7919.231,E2 7919.231} C_VEL
LIN {X 0,Y 251.584,Z 918.976,A -85,B 0,C 180,E1 7916.045,E2 7916.045} C_VEL
LIN {X 0,Y 266.276,Z 903.238,A -85,B 0,C 180,E1 7913.316,E2 7913.316} C_VEL
LIN {X 0,Y 280.933,Z 886.042,A -85,B 0,C 180,E1 7910.991,E2 7910.991} C_VEL
LIN {X 0,Y 294.25,Z 868.443,A -85,B 0,C 180,E1 7909.137,E2 7909.137} C_VEL
LIN {X 0,Y 307.804,Z 848.304,A -85,B 0,C 180,E1 7907.473,E2 7907.473} C_VEL
LIN {X 0,Y 316.865,Z 833.083,A -85,B 0,C 180,E1 7906.444,E2 7906.444} C_VEL
LIN {X 0,Y 310.015,Z 844.928,A -85,B 0,C 180,E1 7905.768,E2 7905.768} C_VEL
LIN {X 0,Y 305.936,Z 851.62,A -85,B 0,C 180,E1 7905.537,E2 7905.537} C_VEL
LIN {X 0,Y 294.529,Z 868.102,A -85,B 0,C 180,E1 7905.517,E2 7905.517} C_VEL
LIN {X 0,Y 290.09,Z 874.11,A -85,B 0,C 180,E1 7905.216,E2 7905.216} C_VEL
LIN {X 0,Y 274.77,Z 893.495,A -85,B 0,C 180,E1 7903.294,E2 7903.294} C_VEL
LIN {X 0,Y 259.987,Z 910.434,A -85,B 0,C 180,E1 7901.111,E2 7901.111} C_VEL
LIN {X 0,Y 244.206,Z 926.71,A -85,B 0,C 180,E1 7898.357,E2 7898.357} C_VEL
LIN {X 0,Y 228.377,Z 941.841,A -85,B 0,C 180,E1 7895.008,E2 7895.008} C_VEL
LIN {X 0,Y 212.786,Z 955.563,A -85,B 0,C 180,E1 7890.939,E2 7890.939} C_VEL
LIN {X 0,Y 197.196,Z 968.5,A -85,B 0,C 180,E1 7885.75,E2 7885.75} C_VEL
LIN {X 0,Y 183.474,Z 979.522,A -85,B 0,C 180,E1 7879.736,E2 7879.736} C_VEL
LIN {X 0,Y 171.96,Z 988.524,A -85,B 0,C 180,E1 7872.878,E2 7872.878} C_VEL
LIN {X 0,Y 162.662,Z 996.157,A -85,B 0,C 180,E1 7864.877,E2 7864.877} C_VEL
LIN {X 0,Y 156.992,Z 1001.297,A -85,B 0,C 180,E1 7857.305,E2 7857.305} C_VEL
LIN {X 0,Y 153.273,Z 1005.536,A -85,B 0,C 180,E1 7848.259,E2 7848.259} C_VEL
LIN {X 0,Y 152.146,Z 1007.589,A -85,B 0,C 180,E1 7840.998,E2 7840.998} C_VEL
LIN {X 0,Y 152.025,Z 1008.46,A -85,B 0,C 180,E1 7834.916,E2 7834.916} C_VEL
LIN {X 0,Y 152.07,Z 1008.534,A -85,B 0,C 180,E1 7829.635,E2 7829.635} C_VEL
LIN {X 0,Y 152.04,Z 1007.881,A -85,B 0,C 180,E1 7823.972,E2 7823.972} C_VEL
LIN {X 0,Y 152.253,Z 1006.345,A -85,B 0,C 180,E1 7817.881,E2 7817.881} C_VEL
LIN {X 0,Y 153.807,Z 1003.053,A -85,B 0,C 180,E1 7809.859,E2 7809.859} C_VEL
LIN {X 0,Y 157.228,Z 998.213,A -85,B 0,C 180,E1 7802.118,E2 7802.118} C_VEL
LIN {X 0,Y 163.1,Z 991.659,A -85,B 0,C 180,E1 7794.397,E2 7794.397} C_VEL
LIN {X 0,Y 171.131,Z 983.394,A -85,B 0,C 180,E1 7787.348,E2 7787.348} C_VEL
LIN {X 0,Y 181.782,Z 972.806,A -85,B 0,C 180,E1 7780.637,E2 7780.637} C_VEL
LIN {X 0,Y 192.641,Z 961.881,A -85,B 0,C 180,E1 7775.444,E2 7775.444} C_VEL
LIN {X 0,Y 204.82,Z 949.025,A -85,B 0,C 180,E1 7770.797,E2 7770.797} C_VEL
LIN {X 0,Y 217.411,Z 934.975,A -85,B 0,C 180,E1 7766.872,E2 7766.872} C_VEL
LIN {X 0,Y 230.496,Z 918.972,A -85,B 0,C 180,E1 7763.467,E2 7763.467} C_VEL
LIN {X 0,Y 243.497,Z 901.664,A -85,B 0,C 180,E1 7760.6,E2 7760.6} C_VEL
LIN {X 0,Y 255.16,Z 884.392,A -85,B 0,C 180,E1 7758.356,E2 7758.356} C_VEL
LIN {X 0,Y 266.757,Z 865.212,A -85,B 0,C 180,E1 7756.385,E2 7756.385} C_VEL
LIN {X 0,Y 276.713,Z 846.634,A -85,B 0,C 180,E1 7754.864,E2 7754.864} C_VEL
LIN {X 0,Y 286.288,Z 826.104,A -85,B 0,C 180,E1 7753.532,E2 7753.532} C_VEL
LIN {X 0,Y 294.843,Z 804.873,A -85,B 0,C 180,E1 7752.443,E2 7752.443} C_VEL
LIN {X 0,Y 302.298,Z 782.356,A -85,B 0,C 180,E1 7751.56,E2 7751.56} C_VEL
LIN {X 0,Y 308.643,Z 758.755,A -85,B 0,C 180,E1 7750.873,E2 7750.873} C_VEL
LIN {X 0,Y 313.11,Z 736.236,A -85,B 0,C 180,E1 7750.358,E2 7750.358} C_VEL
LIN {X 0,Y 317.173,Z 704.32,A -85,B 0,C 180,E1 7749.741,E2 7749.741} C_VEL
LIN {X 0,Y 328.97,Z 597.789,A -85,B 0,C 180,E1 7747.794,E2 7747.794} C_VEL
LIN {X 0,Y 324.567,Z 590.331,A -85,B 0,C 180,E1 7744.062,E2 7744.062} C_VEL
LIN {X 0,Y 321.662,Z 585.746,A -85,B 0,C 180,E1 7741.068,E2 7741.068} C_VEL
LIN {X 0,Y 319.307,Z 581.79,A -85,B 0,C 180,E1 7738.025,E2 7738.025} C_VEL
LIN {X 0,Y 316.866,Z 577.642,A -85,B 0,C 180,E1 7733.635,E2 7733.635} C_VEL
LIN {X 0,Y 316.122,Z 576.818,A -85,B 0,C 180,E1 7731.817,E2 7731.817} C_VEL
LIN {X 0,Y 315.027,Z 575.632,A -85,B 0,C 180,E1 7726.041,E2 7726.041} C_VEL
LIN {X 0,Y 315.57,Z 576.355,A -85,B 0,C 180,E1 7721.144,E2 7721.144} C_VEL
LIN {X 0,Y 316.876,Z 577.53,A -85,B 0,C 180,E1 7717.652,E2 7717.652} C_VEL
LIN {X 0,Y 319.962,Z 582.811,A -85,B 0,C 180,E1 7712.35,E2 7712.35} C_VEL
LIN {X 0,Y 322.816,Z 587.523,A -85,B 0,C 180,E1 7708.955,E2 7708.955} C_VEL
LIN {X 0,Y 325.832,Z 592.555,A -85,B 0,C 180,E1 7706.048,E2 7706.048} C_VEL
LIN {X 0,Y 328.655,Z 597.401,A -85,B 0,C 180,E1 7703.709,E2 7703.709} C_VEL
LIN {X 0,Y 314.559,Z 722.031,A -85,B 0,C 180,E1 7701.454,E2 7701.454} C_VEL
LIN {X 0,Y 310.21,Z 745.8,A -85,B 0,C 180,E1 7700.91,E2 7700.91} C_VEL
LIN {X 0,Y 304.84,Z 767.939,A -85,B 0,C 180,E1 7700.238,E2 7700.238} C_VEL
LIN {X 0,Y 298.24,Z 789.11,A -85,B 0,C 180,E1 7699.395,E2 7699.395} C_VEL
LIN {X 0,Y 289.949,Z 811.393,A -85,B 0,C 180,E1 7698.268,E2 7698.268} C_VEL
LIN {X 0,Y 281.01,Z 831.582,A -85,B 0,C 180,E1 7696.974,E2 7696.974} C_VEL
